    CASE VI_First_Fault_Source OF
        1: L_First_Fault_Source_Text := 'Heating';
        2: L_First_Fault_Source_Text := 'DHW';
        3: L_First_Fault_Source_Text := 'Ventilation';
        4: L_First_Fault_Source_Text := 'Lighting';
        5: L_First_Fault_Source_Text := 'Access';
        ELSE L_First_Fault_Source_Text := 'Unknown';
    END_CASE;

    L_Pending_Alarms[L_Pending_Count].Message := CONCAT('Diagnostics root cause: ', CONCAT(L_First_Fault_Source_Text, CONCAT(' / ', L_First_Fault_Type_Text)));
    L_Pending_Alarms[L_Pending_Count].Severity := E_ALERT_PRIORITY.ALERT_PRIORITY_HIGH;
    L_Pending_Alarms[L_Pending_Count].Is_Active := TRUE;
    L_Pending_Alarms[L_Pending_Count].Is_Acknowledged := FALSE;
END_IF;

FOR L_j := 1 TO GVL_CONSTANTS.C_MAX_BOILERS DO
    IF R_Trig_Boiler[L_j].Q AND L_Pending_Count < 10 THEN
        L_Pending_Count := L_Pending_Count + 1;
        L_Pending_Alarms[L_Pending_Count].Timestamp_MS := VI_System_Time_MS;
        L_Pending_Alarms[L_Pending_Count].Source := 'Boiler';
        L_Pending_Alarms[L_Pending_Count].Source_ID := TO_BYTE(L_j);
        L_Pending_Alarms[L_Pending_Count].Message := CONCAT('Авария котла №', INT_TO_STRING(L_j));
        L_Pending_Alarms[L_Pending_Count].Severity := E_ALERT_PRIORITY.ALERT_PRIORITY_HIGH;
        L_Pending_Alarms[L_Pending_Count].Is_Active := TRUE;
        L_Pending_Alarms[L_Pending_Count].Is_Acknowledged := FALSE;
    END_IF;
END_FOR;



// Обработка очереди новых тревог с учетом приоритетов
FOR L_i := 1 TO L_Pending_Count DO

    L_Target_Slot := 0;
    
    // 1. Ищем пустой слот
    FOR L_k := 1 TO GVL_CONSTANTS.C_MAX_ALARMS DO
        IF VO_Alarm_List[L_k].ID = 0 THEN
            L_Target_Slot := L_k;
            EXIT;
        END_IF;
    END_FOR;
    
    // 2. Ищем квитированную тревогу с наименьшим приоритетом
    IF L_Target_Slot = 0 THEN
        L_Min_Pri := 999;
        FOR L_k := 1 TO GVL_CONSTANTS.C_MAX_ALARMS DO
            IF VO_Alarm_List[L_k].Is_Acknowledged AND TO_INT(VO_Alarm_List[L_k].Severity) < L_Min_Pri THEN
                L_Min_Pri := TO_INT(VO_Alarm_List[L_k].Severity);
                L_Target_Slot := L_k;
            END_IF;
        END_FOR;
    END_IF;
    
    // 3. Ищем неквитированную тревогу с наименьшим приоритетом (если он ниже добавляемой)
    IF L_Target_Slot = 0 THEN
        L_Min_Pri := 999;
        FOR L_k := 1 TO GVL_CONSTANTS.C_MAX_ALARMS DO
            IF TO_INT(VO_Alarm_List[L_k].Severity) < L_Min_Pri AND TO_INT(VO_Alarm_List[L_k].Severity) < TO_INT(L_Pending_Alarms[L_i].Severity) THEN
                L_Min_Pri := TO_INT(VO_Alarm_List[L_k].Severity);
                L_Target_Slot := L_k;
            END_IF;
        END_FOR;
    END_IF;
    
    IF L_Target_Slot = 0 THEN 
        // Буфер полон критических неквитированных тревог. Не затираем!
        CONTINUE; 
    END_IF;
    
    VO_Alarm_List[L_Target_Slot] := L_Pending_Alarms[L_i];
    VO_Alarm_List[L_Target_Slot].ID := VIO_Next_Alarm_ID;
    VIO_Next_Alarm_ID := VIO_Next_Alarm_ID + 1;
    IF VIO_Next_Alarm_ID = 0 THEN VIO_Next_Alarm_ID := 1; END_IF;
    IF NOT L_Event_Pulse_Latched THEN
        VO_Event_Pulse := TRUE;
        VO_Event_Code := 1203;
        VO_Event_Value := TO_REAL(VO_Alarm_List[L_Target_Slot].Severity);
        L_Event_Pulse_Latched := TRUE;
    END_IF;
END_FOR;

// 3. Обновление статуса существующих тревог (ушли ли они?)
FOR L_i := 1 TO GVL_CONSTANTS.C_MAX_ALARMS DO
    IF VO_Alarm_List[L_i].ID <> 0 THEN
        IF VO_Alarm_List[L_i].Source = 'Gas' THEN VO_Alarm_List[L_i].Is_Active := VI_Gas_Alarm;
        ELSIF VO_Alarm_List[L_i].Source = 'Fire' THEN VO_Alarm_List[L_i].Is_Active := VI_Fire_Alarm;
        ELSIF VO_Alarm_List[L_i].Source = 'Flood' THEN VO_Alarm_List[L_i].Is_Active := VI_Flood_Alarm;
        ELSIF VO_Alarm_List[L_i].Source = 'Security' THEN VO_Alarm_List[L_i].Is_Active := VI_Security_Alarm;
        ELSIF VO_Alarm_List[L_i].Source = 'Diagnostics' THEN VO_Alarm_List[L_i].Is_Active := VI_First_Fault_Active;
        ELSIF VO_Alarm_List[L_i].Source = 'Boiler' THEN 
            IF TO_INT(VO_Alarm_List[L_i].Source_ID) >= 1 AND TO_INT(VO_Alarm_List[L_i].Source_ID) <= GVL_CONSTANTS.C_MAX_BOILERS THEN
                VO_Alarm_List[L_i].Is_Active := VI_Boiler_Errors[TO_INT(VO_Alarm_List[L_i].Source_ID)];
            END_IF;
        END_IF;
    END_IF;
END_FOR;

// 4. Квитирование тревог
IF VI_Acknowledge_All THEN
    FOR L_i := 1 TO GVL_CONSTANTS.C_MAX_ALARMS DO
        IF VO_Alarm_List[L_i].ID <> 0 THEN
            VO_Alarm_List[L_i].Is_Acknowledged := TRUE;
        END_IF;
    END_FOR;

    IF NOT L_Event_Pulse_Latched THEN
        VO_Event_Pulse := TRUE;
        VO_Event_Code := 1201;
        VO_Event_Value := TO_REAL(VO_Unacked_Count);
        L_Event_Pulse_Latched := TRUE;
    END_IF;
END_IF;

// 4.5 Автоквитирование некритичных тревог, если они больше не активны
FOR L_i := 1 TO GVL_CONSTANTS.C_MAX_ALARMS DO
    IF VO_Alarm_List[L_i].ID <> 0 AND NOT VO_Alarm_List[L_i].Is_Active AND NOT VO_Alarm_List[L_i].Is_Acknowledged THEN
        IF VO_Alarm_List[L_i].Severity <> E_ALERT_PRIORITY.ALERT_PRIORITY_CRITICAL THEN
            VO_Alarm_List[L_i].Is_Acknowledged := TRUE;
        END_IF;
    END_IF;
END_FOR;

// 5. Очистка списка (удаление неактивных И квитированных тревог)
// В кольцевом буфере мы просто помечаем слот как пустой (ID = 0), без сдвига массива
FOR L_i := 1 TO GVL_CONSTANTS.C_MAX_ALARMS DO
    IF VO_Alarm_List[L_i].ID <> 0 AND NOT VO_Alarm_List[L_i].Is_Active AND VO_Alarm_List[L_i].Is_Acknowledged THEN
        // Удаляем тревогу
        VO_Alarm_List[L_i].ID := 0;
        IF NOT L_Event_Pulse_Latched THEN
            VO_Event_Pulse := TRUE;
            VO_Event_Code := 1202;
            VO_Event_Value := 0.0;
            L_Event_Pulse_Latched := TRUE;
        END_IF;
    END_IF;
END_FOR;


// 6. Подсчет статистики и формирование глобальных флагов
VO_Global_Critical := FALSE;
VO_Global_Warning := FALSE;
VO_Siren_Active := FALSE;
VO_Active_Count := 0;
VO_Unacked_Count := 0;

FOR L_i := 1 TO GVL_CONSTANTS.C_MAX_ALARMS DO
    IF VO_Alarm_List[L_i].ID <> 0 THEN
        IF VO_Alarm_List[L_i].Is_Active THEN
            VO_Active_Count := VO_Active_Count + 1;
        END_IF;
        
        IF NOT VO_Alarm_List[L_i].Is_Acknowledged THEN
            VO_Unacked_Count := VO_Unacked_Count + 1;
            
            IF VO_Alarm_List[L_i].Severity = E_ALERT_PRIORITY.ALERT_PRIORITY_CRITICAL THEN
                VO_Global_Critical := TRUE;
                // Сирена работает только для неквитированных критических тревог, если не включен Mute
                IF NOT VI_Mute_Siren THEN
                    VO_Siren_Active := TRUE;
                END_IF;
            ELSIF VO_Alarm_List[L_i].Severity = E_ALERT_PRIORITY.ALERT_PRIORITY_HIGH THEN
                VO_Global_Warning := TRUE;
            END_IF;
        END_IF;
    END_IF;
END_FOR;
// >>> BULK_SYNC_ANCHOR: FB_Alarm_Manager <<<
          
END_FUNCTION_BLOCK

FUNCTION_BLOCK FB_Distributed_Recovery_Lock_Runtime
  VAR_INPUT
    VI_Enable : BOOL;
    VI_System_Time_MS : UDINT;
  END_VAR
  VAR
    L_Lock : ST_Distributed_Recovery_Lock;
    L_Finalized_Runtime_Continuity : BOOL;
  END_VAR

            IF NOT VI_Enable THEN
    GVL_Distributed_Recovery_Lock.G_Runtime_Valid := FALSE;
    RETURN;
END_IF;

L_Lock := GVL_Distributed_Recovery_Lock.G_Recovery_Lock;

L_Lock.Runtime_System_Time_MS := VI_System_Time_MS;
L_Lock.Lock_Valid := TRUE;

// Finalized runtime continuity proof chain.
L_Finalized_Runtime_Continuity :=
    GVL_SEMANTIC_PROGRESS.Semantic_Forward_Progress_Valid
    AND GVL_SEMANTIC_PROGRESS.Semantic_Execution_Continuity_OK
    AND NOT GVL_SEMANTIC_PROGRESS.Semantic_Progress_Lease_Expired
    AND NOT GVL_SEMANTIC_PROGRESS.Semantic_Progress_Quarantine_Active
    AND GVL_RUNTIME_SNAPSHOT.Snapshot_Frozen
    AND GVL_RUNTIME_SNAPSHOT.Snapshot_Publication_Allowed
    AND GVL_RUNTIME_SNAPSHOT.Snapshot_Copy_Valid
    AND GVL_RUNTIME_SNAPSHOT.Snapshot_Isolation_Valid
    AND NOT GVL_RUNTIME_SNAPSHOT.Snapshot_Mutation_Detected
    AND GVL_DISTRIBUTED_SNAPSHOT.Distributed_Publication_Reconciled
    AND GVL_DISTRIBUTED_SNAPSHOT.Distributed_Publication_Freeze_Valid
    AND GVL_DISTRIBUTED_SNAPSHOT.Distributed_Snapshot_Consistent
    AND GVL_DISTRIBUTED_COMMIT.Distributed_Commit_Valid
    AND GVL_DISTRIBUTED_COMMIT.Publication_Prepare_Valid
    AND GVL_DISTRIBUTED_COMMIT.Publication_Commit_Confirmed
    AND NOT GVL_DISTRIBUTED_COMMIT.Peer_Commit_Mismatch
    AND NOT GVL_DISTRIBUTED_COMMIT.Commit_Lease_Expired
    AND GVL_OUTPUT_EPOCH.Output_Publication_Valid
    AND GVL_OUTPUT_EPOCH.Output_Runtime_Epoch_Valid
    AND NOT GVL_OUTPUT_EPOCH.Output_Lease_Expired
    AND NOT GVL_OUTPUT_EPOCH.Output_Forced_Safe_Decay
    AND GVL_COMMAND_VERIFY.PreOutput_Barrier_OK
    AND NOT GVL_COMMAND_VERIFY.PreOutput_Block_IO;

// Cluster-exclusive recovery execution lock.
IF GVL_Distributed_Runtime.G_Split_Brain_Suspected
   OR GVL_Distributed_Projection_Ownership.G_Any_Ownership_Conflict
   OR GVL_Runtime_Sessions.G_Any_Stale_Session
   OR NOT L_Finalized_Runtime_Continuity THEN

    L_Lock.Lock_Conflict := TRUE;
    L_Lock.Distributed_Execution_Allowed := FALSE;

    GVL_Distributed_Recovery_Lock.G_Recovery_Execution_Blocked := TRUE;
    GVL_Distributed_Recovery_Lock.G_Rollback_Execution_Blocked := TRUE;
    GVL_Distributed_Recovery_Lock.G_Reopen_Execution_Blocked := TRUE;

    L_Lock.Status_Code := 3;
    L_Lock.Status_Text :=
        'Distributed recovery execution locked';

ELSE

    L_Lock.Recovery_Lock_Active := TRUE;
    L_Lock.Distributed_Execution_Allowed := TRUE;

    GVL_Distributed_Recovery_Lock.G_Recovery_Execution_Blocked := FALSE;
    GVL_Distributed_Recovery_Lock.G_Rollback_Execution_Blocked := FALSE;
    GVL_Distributed_Recovery_Lock.G_Reopen_Execution_Blocked := FALSE;

    L_Lock.Status_Code := 0;
    L_Lock.Status_Text :=
        'Distributed recovery lock healthy';

END_IF;

GVL_Distributed_Recovery_Lock.G_Recovery_Lock := L_Lock;

GVL_Distributed_Recovery_Lock.G_Runtime_Valid := TRUE;
GVL_Distributed_Recovery_Lock.G_Last_Update_MS :=
    VI_System_Time_MS;

GVL_Distributed_Recovery_Lock.G_Status_Code :=
    L_Lock.Status_Code;

GVL_Distributed_Recovery_Lock.G_Status_Text :=
    L_Lock.Status_Text;
          
END_FUNCTION_BLOCK

FUNCTION_BLOCK FB_Heating_Predictive_Controller
  VAR
    L_i : INT;
    L_Time_To_Heat : UDINT;
    L_Time_To_Comfort : UDINT;
    L_Now_TOD : UDINT;
  END_VAR

            // ==============================================================================
// Ownership note
// ------------------------------------------------------------------------------
// This block owns predictive preheat decision only.
// It does NOT modify thermal demand. Thermal demand is owned by
// FB_Heating_Thermal_Model and may be interpreted by downstream advisory layers.
// ==============================================================================

L_Now_TOD := GVL_TIME_SERVICE.G_Time_Of_Day_MS;

FOR L_i := 1 TO GVL_CONSTANTS.C_MAX_ZONES DO

    L_Time_To_Heat := GVL_HEATING_POLICY.G_Zone_Time_To_Heat_MS[L_i];
    L_Time_To_Comfort := GVL_HEATING_POLICY.G_Zone_Comfort_Time_MS[L_i];

    // Predictive preheat decision.
    IF GVL_HEATING_POLICY.G_Zone_Schedule_Enabled[L_i] THEN

        IF L_Time_To_Comfort > L_Now_TOD THEN
            IF (L_Time_To_Comfort - L_Now_TOD) <= L_Time_To_Heat THEN
                GVL_HEATING_POLICY.G_Zone_Preheat_Needed[L_i] := TRUE;
            ELSE
                GVL_HEATING_POLICY.G_Zone_Preheat_Needed[L_i] := FALSE;
            END_IF;
        END_IF;

    END_IF;

    // Confidence gating.
    IF GVL_HEATING_POLICY.G_Zone_Thermal_Model_Confidence[L_i] < 0.1 THEN
        GVL_HEATING_POLICY.G_Zone_Preheat_Needed[L_i] := FALSE;
    END_IF;

END_FOR;
          
END_FUNCTION_BLOCK

FUNCTION_BLOCK FB_System_Coordinator
  VAR_INPUT
    VI_Fire_Latched : BOOL;
    VI_Gas_Latched : BOOL;
    VI_Leak_Latched : BOOL;
    VI_IO_Degraded : BOOL;
    VI_Ownership_Violation : BOOL;
    VI_Behavior_Mode : E_Behavior_Mode;
  END_VAR
  VAR_OUTPUT
    VO_Block_Heating : BOOL;
    VO_Block_Ventilation : BOOL;
    VO_Block_Lighting : BOOL;
    VO_Block_Sockets : BOOL;
    VO_System_Degraded : BOOL;
    VO_Code : UDINT;
  END_VAR

            // reset
VO_Block_Heating := FALSE;
VO_Block_Ventilation := FALSE;
VO_Block_Lighting := FALSE;
VO_Block_Sockets := FALSE;
VO_System_Degraded := FALSE;
VO_Code := 0;

// FIRE has highest priority. Safety-stop ownership remains in PRG_Safety.
IF VI_Fire_Latched THEN
    VO_Block_Heating := TRUE;
    VO_Block_Ventilation := TRUE;
    VO_Block_Sockets := TRUE;
    VO_Code := 100;
    RETURN;
END_IF;

// GAS has higher priority than behavior mode.
IF VI_Gas_Latched THEN
    VO_Block_Heating := TRUE;
    VO_Block_Lighting := TRUE;
    VO_Block_Sockets := TRUE;
    VO_Code := 200;
    RETURN;
END_IF;

// LEAK blocks heating but does not suppress later degradation/mode overlays.
IF VI_Leak_Latched THEN
    VO_Block_Heating := TRUE;
    VO_Code := 300;
END_IF;

// IO degraded blocks heating and marks system degraded.
IF VI_IO_Degraded THEN
    VO_System_Degraded := TRUE;
    VO_Block_Heating := TRUE;
    IF VO_Code = 0 THEN
        VO_Code := 400;
    END_IF;
END_IF;

// Ownership violation marks system degraded. Test/result handler owns any safe-stop reaction.
IF VI_Ownership_Violation THEN
    VO_System_Degraded := TRUE;
    IF VO_Code = 0 THEN
        VO_Code := 500;
    END_IF;
END_IF;

// Behavior mode overlays. These are lower priority than safety/system faults.
CASE VI_Behavior_Mode OF
    BEHAVIOR_AWAY:
        VO_Block_Lighting := TRUE;
        VO_Block_Sockets := TRUE;
        IF VO_Code = 0 THEN
            VO_Code := 600;
        END_IF;

    BEHAVIOR_NIGHT:
        VO_Block_Lighting := TRUE;
        IF VO_Code = 0 THEN
            VO_Code := 700;
        END_IF;

    BEHAVIOR_MAINTENANCE:
        VO_Block_Heating := TRUE;
        VO_Block_Ventilation := TRUE;
        IF VO_Code = 0 THEN
            VO_Code := 800;
        END_IF;
ELSE
        // No fallback required
END_CASE;
          
END_FUNCTION_BLOCK

FUNCTION_BLOCK FB_Water_Isolation_Path_Resolver
  VAR_INPUT
    VI_Enable : BOOL;
    VI_System_Time_MS : UDINT;
  END_VAR
  VAR
    L_i : INT;
    L_Edge : ST_Water_Hydraulic_Topology_Edge;
    L_Path : ST_Water_Isolation_Path_Runtime_State;
    L_Validation : ST_Water_Topology_Validation_State;
    L_Any_Shared_Trunk : BOOL;
    L_Any_Conflict : BOOL;
    L_Any_Fallback : BOOL;
  END_VAR

            IF NOT VI_Enable THEN
    GVL_Water_Hydraulic_Graph.G_Runtime_Valid := FALSE;
    RETURN;
END_IF;

FOR L_i := 1 TO GVL_CONSTANTS.C_MAX_FLOOD_SENSORS DO

    L_Validation :=
        GVL_Water_Topology_Validation.G_Validation_State[L_i];

    // Graph edge publication.
    L_Edge := (Runtime_Valid := TRUE);

    L_Edge.Edge_Id := TO_UINT(L_i);

    L_Edge.Upstream_Segment_Id :=
        GVL_Water_Hydraulic_Topology.G_Topology_Node[L_i].Hydraulic_Segment_Id;

    L_Edge.Downstream_Segment_Id :=
        GVL_Water_Hydraulic_Topology.G_Topology_Node[L_i].Hydraulic_Zone_Id;

    L_Edge.Isolation_Group_Id :=
        GVL_Water_Hydraulic_Topology.G_Topology_Node[L_i].Isolation_Group_Id;

    L_Edge.Valve_Group_Id :=
        GVL_Water_Hydraulic_Topology.G_Topology_Node[L_i].Valve_Group_Id;

    // Shared trunk semantics.
    IF L_Edge.Valve_Group_Id = 3 THEN
        L_Edge.Shared_Trunk := TRUE;
        L_Edge.Cross_Zone_Dependency := TRUE;
    END_IF;

    L_Edge.Dependency_Valid :=
        L_Validation.Topology_Valid;

    L_Edge.Dependency_Ambiguous :=
        L_Validation.Topology_Ambiguous;

    L_Edge.Selective_Isolation_Allowed :=
        L_Validation.Selective_Isolation_Allowed;

    L_Edge.Global_Fallback_Required :=
        L_Validation.Global_Fallback_Required;

    // Isolation path runtime.
    L_Path := (Runtime_Valid := TRUE);

    L_Path.Runtime_System_Time_MS :=
        VI_System_Time_MS;

    L_Path.Sensor_Id := TO_UINT(L_i);

    L_Path.Isolation_Path_Valid :=
        L_Edge.Dependency_Valid;

    L_Path.Isolation_Path_Ambiguous :=
        L_Edge.Dependency_Ambiguous;

    L_Path.Active_Isolation_Group_Id :=
        L_Edge.Isolation_Group_Id;

    L_Path.Active_Valve_Group_Id :=
        L_Edge.Valve_Group_Id;

    L_Path.Shared_Trunk_Impact :=
        L_Edge.Shared_Trunk;

    L_Path.Cross_Zone_Impact :=
        L_Edge.Cross_Zone_Dependency;

    L_Path.Selective_Isolation_Allowed :=
        L_Edge.Selective_Isolation_Allowed;

    L_Path.Global_Fallback_Required :=
        L_Edge.Global_Fallback_Required;

    // Multi-valve/shared-trunk path.
    IF L_Path.Shared_Trunk_Impact THEN
        L_Path.Multi_Valve_Path := TRUE;
    END_IF;

    // Conflict detection.
    IF L_Path.Isolation_Path_Ambiguous THEN
        L_Path.Conflict_Detected := TRUE;
    END_IF;

    // Conservative escalation.
    IF L_Path.Conflict_Detected THEN
        L_Path.Global_Fallback_Required := TRUE;
        L_Path.Selective_Isolation_Allowed := FALSE;

        L_Path.Status_Code := 2;
        L_Path.Status_Text :=
            'Isolation path conflict detected';

    ELSIF L_Path.Shared_Trunk_Impact THEN
        L_Path.Status_Code := 1;
        L_Path.Status_Text :=
            'Shared trunk isolation path active';

    ELSE
        L_Path.Status_Code := 0;
        L_Path.Status_Text :=
            'Isolation path resolved';
    END_IF;

    GVL_Water_Hydraulic_Graph.G_Topology_Edge[L_i] :=
        L_Edge;

    GVL_Water_Hydraulic_Graph.G_Isolation_Path[L_i] :=
        L_Path;

    L_Any_Shared_Trunk :=
        L_Any_Shared_Trunk
        OR L_Path.Shared_Trunk_Impact;

    L_Any_Conflict :=
        L_Any_Conflict
        OR L_Path.Conflict_Detected;

    L_Any_Fallback :=
        L_Any_Fallback
        OR L_Path.Global_Fallback_Required;

END_FOR;

GVL_Water_Hydraulic_Graph.G_Any_Shared_Trunk :=
    L_Any_Shared_Trunk;

GVL_Water_Hydraulic_Graph.G_Any_Conflict :=
    L_Any_Conflict;

GVL_Water_Hydraulic_Graph.G_Any_Global_Fallback_Required :=
    L_Any_Fallback;

GVL_Water_Hydraulic_Graph.G_Runtime_Valid := TRUE;
GVL_Water_Hydraulic_Graph.G_Last_Update_MS := VI_System_Time_MS;

IF L_Any_Conflict THEN
    GVL_Water_Hydraulic_Graph.G_Status_Code := 2;
    GVL_Water_Hydraulic_Graph.G_Status_Text :=
        'Hydraulic graph conflicts detected';
ELSIF L_Any_Shared_Trunk THEN
    GVL_Water_Hydraulic_Graph.G_Status_Code := 1;
    GVL_Water_Hydraulic_Graph.G_Status_Text :=
        'Shared trunk governance active';
ELSE
    GVL_Water_Hydraulic_Graph.G_Status_Code := 0;
    GVL_Water_Hydraulic_Graph.G_Status_Text :=
        'Hydraulic graph runtime healthy';
END_IF;
          
END_FUNCTION_BLOCK

FUNCTION_BLOCK FB_Ownership_Watchdog
  VAR_INPUT
    VI_Gas_Level : REAL;
    VI_Gas_Alarm : BOOL;
    VI_Leak_Alarm : BOOL;
    VI_Smoke_Alarm : BOOL;
  END_VAR
  VAR_OUTPUT
    VO_Ownership_Violation : BOOL;
  END_VAR
  VAR
    L_Last_Gas_Alarm : BOOL;
    L_Last_Leak_Alarm : BOOL;
    L_Last_Smoke_Alarm : BOOL;
  END_VAR

            VO_Ownership_Violation := FALSE;

// Gas: signal present, alarm disappeared
IF (VI_Gas_Level > 20.0) AND L_Last_Gas_Alarm AND (NOT VI_Gas_Alarm) THEN
    VO_Ownership_Violation := TRUE;
END_IF;

// Leak: once latched should not drop instantly
IF L_Last_Leak_Alarm AND (NOT VI_Leak_Alarm) THEN
    VO_Ownership_Violation := TRUE;
END_IF;

// Smoke: same rule
IF L_Last_Smoke_Alarm AND (NOT VI_Smoke_Alarm) THEN
    VO_Ownership_Violation := TRUE;
END_IF;

L_Last_Gas_Alarm := VI_Gas_Alarm;
L_Last_Leak_Alarm := VI_Leak_Alarm;
L_Last_Smoke_Alarm := VI_Smoke_Alarm;
          
END_FUNCTION_BLOCK

FUNCTION_BLOCK FB_Valve_Test_Manager
  VAR_INPUT
    VI_System_Time_MS : UDINT;
    VI_IsActivePLC : BOOL;
  END_VAR
  VAR_OUTPUT
    VO_Test_Active : BOOL;
    VO_Current_Valve : INT;
    VO_Valve_Cmd : ARRAY[1..GVL_CONSTANTS.C_MAX_MANIFOLDS] OF BOOL;
    VO_Test_Results : ARRAY[1..GVL_CONSTANTS.C_MAX_MANIFOLDS] OF BOOL;
    VO_Status_Msg : STRING(200);
  END_VAR
  VAR_IN_OUT
    VI_Valve_Currents : ARRAY[1..GVL_CONSTANTS.C_MAX_MANIFOLDS] OF REAL;
    VI_Valve_End_Switches : ARRAY[1..GVL_CONSTANTS.C_MAX_MANIFOLDS] OF BOOL;
    VI_Config : ARRAY[1..GVL_CONSTANTS.C_MAX_MANIFOLDS] OF ST_Valve_Test_Config;
  END_VAR
  VAR
    L_State : INT;
    L_Current_Valve : INT := 1;
    L_Test_Start_Time : UDINT;
    L_Last_Test_Time : ARRAY[1..GVL_CONSTANTS.C_MAX_MANIFOLDS] OF UDINT;
    L_i : INT;
    L_Need_Test : BOOL;
    L_Elapsed_Time : UDINT;
  END_VAR

            IF NOT VI_IsActivePLC THEN RETURN; END_IF;

CASE L_State OF
    0: // Ожидание
        VO_Test_Active := FALSE;
        L_Need_Test := FALSE;
        
        // Поиск клапана, которому нужен тест (раз в неделю)
        FOR L_i := 1 TO GVL_CONSTANTS.C_MAX_MANIFOLDS DO
            IF VI_Config[L_i].enabled AND ((VI_System_Time_MS - L_Last_Test_Time[L_i]) > (VI_Config[L_i].test_interval_days * 86400000)) THEN
                L_Current_Valve := L_i;
                L_Need_Test := TRUE;
                EXIT;
            END_IF;
        END_FOR;
        
        IF L_Need_Test THEN
            L_State := 1;
            L_Test_Start_Time := VI_System_Time_MS;
            VO_Test_Active := TRUE;
            VO_Current_Valve := L_Current_Valve;
            VO_Valve_Cmd[L_Current_Valve] := TRUE; // Открываем
            VO_Status_Msg := CONCAT('ТЕСТ КЛАПАНА ', INT_TO_STRING(L_Current_Valve));
            VO_Test_Results[L_Current_Valve] := TRUE; // Сброс результата
        END_IF;
        
    1: // Тестирование (ожидание открытия)
        L_Elapsed_Time := (VI_System_Time_MS - L_Test_Start_Time);
        
        IF VI_Valve_End_Switches[L_Current_Valve] THEN
            // Концевик сработал до истечения таймаута
            // Проверка тока
            IF ABS(VI_Valve_Currents[L_Current_Valve] - VI_Config[L_Current_Valve].Nominal_Current) > (VI_Config[L_Current_Valve].Nominal_Current * 0.2) THEN
                VO_Test_Results[L_Current_Valve] := FALSE; // Ошибка по току
            END_IF;
            
            GVL_Retain.G_Valve_Test_Results[L_Current_Valve] := VO_Test_Results[L_Current_Valve];
            
            VO_Valve_Cmd[L_Current_Valve] := FALSE; // Закрываем
            L_Test_Start_Time := VI_System_Time_MS; // Перезапускаем таймер для проверки закрытия
            L_State := 2;
        ELSIF L_Elapsed_Time > TO_UDINT(VI_Config[L_Current_Valve].nominal_close_time_sec * 1000.0) THEN
            // Таймаут открытия (заклинивание)
            VO_Test_Results[L_Current_Valve] := FALSE; 
            GVL_Retain.G_Valve_Test_Results[L_Current_Valve] := FALSE;
            VO_Status_Msg := CONCAT('ОШИБКА: ЗАКЛИНИВАНИЕ КЛАПАНА ', INT_TO_STRING(L_Current_Valve));
            
            VO_Valve_Cmd[L_Current_Valve] := FALSE; // Закрываем
            L_Test_Start_Time := VI_System_Time_MS; // Перезапускаем таймер
            L_State := 2;
        END_IF;
        
    2: // Ожидание закрытия
        L_Elapsed_Time := (VI_System_Time_MS - L_Test_Start_Time);
        
        IF NOT VI_Valve_End_Switches[L_Current_Valve] THEN
            // Концевик разомкнулся (клапан закрыт)
            L_Last_Test_Time[L_Current_Valve] := VI_System_Time_MS;
            L_State := 0;
            IF VO_Test_Results[L_Current_Valve] THEN
                VO_Status_Msg := 'ТЕСТ ЗАВЕРШЕН УСПЕШНО';
            END_IF;
        ELSIF L_Elapsed_Time > TO_UDINT(VI_Config[L_Current_Valve].nominal_close_time_sec * 1000.0) THEN
            // Таймаут закрытия (заклинивание)
            VO_Test_Results[L_Current_Valve] := FALSE; 
            GVL_Retain.G_Valve_Test_Results[L_Current_Valve] := FALSE;
            VO_Status_Msg := CONCAT('ОШИБКА: НЕ ЗАКРЫЛСЯ КЛАПАН ', INT_TO_STRING(L_Current_Valve));
            
            L_Last_Test_Time[L_Current_Valve] := VI_System_Time_MS;
            L_State := 0;
        END_IF;
ELSE
        // No fallback required
END_CASE;
          
END_FUNCTION_BLOCK

FUNCTION_BLOCK FB_PID_Controller
  VAR_INPUT
    VI_SetPoint : REAL;
    VI_ProcessValue : REAL;
    VI_Kp : REAL;
    VI_Tn : REAL;
    VI_Tv : REAL;
    VI_Y_Min : REAL := REAL#0.0;
    VI_Y_Max : REAL := REAL#100.0;
    VI_Manual_Mode : BOOL;
    VI_Manual_Value : REAL;
    VI_Deadband : REAL := REAL#0.1;
    VI_Cycle_Time_S : REAL := REAL#0.01;
    VI_Reset : BOOL;
  END_VAR
  VAR_OUTPUT
    VO_Output : REAL;
    VO_Error : REAL;
    VO_Limiting : BOOL;
  END_VAR
  VAR
    L_Integral_Sum : REAL;
    L_Prev_Error : REAL;
    L_Derivative : REAL;
    L_P_Term : REAL;
    L_I_Candidate : REAL;
    L_D_Term : REAL;
    L_Output_Predicted : REAL;
    L_Output_Raw : REAL;
    L_Cycle_Time_Safe : REAL;
  END_VAR

            L_Cycle_Time_Safe := VI_Cycle_Time_S;
IF L_Cycle_Time_Safe <= REAL#0.0 THEN
    L_Cycle_Time_Safe := REAL#0.01;
END_IF;

VO_Error := VI_SetPoint - VI_ProcessValue;
IF ABS(VO_Error) < VI_Deadband THEN
    VO_Error := REAL#0.0;
END_IF;

IF VI_Reset THEN
    L_Integral_Sum := REAL#0.0;
    L_Prev_Error := REAL#0.0;
    VO_Output := LIMIT(VI_Y_Min, REAL#0.0, VI_Y_Max);
    VO_Limiting := FALSE;
    RETURN;
END_IF;

L_P_Term := VI_Kp * VO_Error;

IF VI_Tv > REAL#0.0 THEN
    L_Derivative := (VO_Error - L_Prev_Error) / L_Cycle_Time_Safe;
    L_D_Term := VI_Kp * VI_Tv * L_Derivative;
ELSE
    L_Derivative := REAL#0.0;
    L_D_Term := REAL#0.0;
END_IF;

IF VI_Manual_Mode THEN
    VO_Output := LIMIT(VI_Y_Min, VI_Manual_Value, VI_Y_Max);
    L_Integral_Sum := VO_Output - L_P_Term - L_D_Term;
    L_Prev_Error := VO_Error;
    VO_Limiting := (VO_Output <= VI_Y_Min) OR (VO_Output >= VI_Y_Max);
    RETURN;
END_IF;

IF VI_Tn > REAL#0.0 THEN
    L_I_Candidate := L_Integral_Sum + ((VI_Kp / VI_Tn) * VO_Error * L_Cycle_Time_Safe);
ELSE
    L_I_Candidate := L_Integral_Sum;
END_IF;

L_Output_Predicted := L_P_Term + L_I_Candidate + L_D_Term;

// Anti-windup: accept the new integral only if it does not push the output farther into saturation.
IF VI_Tn > REAL#0.0 THEN
    IF (L_Output_Predicted > VI_Y_Max) AND (VO_Error > REAL#0.0) THEN
        // hold integral
    ELSIF (L_Output_Predicted < VI_Y_Min) AND (VO_Error < REAL#0.0) THEN
        // hold integral
    ELSE
        L_Integral_Sum := L_I_Candidate;
    END_IF;
END_IF;

L_Output_Raw := L_P_Term + L_Integral_Sum + L_D_Term;
VO_Output := LIMIT(VI_Y_Min, L_Output_Raw, VI_Y_Max);
VO_Limiting := (L_Output_Raw > VI_Y_Max) OR (L_Output_Raw < VI_Y_Min);
L_Prev_Error := VO_Error;

// >>> BULK_SYNC_ANCHOR: FB_PID_Controller <<<
          
END_FUNCTION_BLOCK

FUNCTION_BLOCK FB_ADS_Runtime_Adapter
  VAR_INPUT
    VI_Enable : BOOL;
    VI_System_Time_MS : UDINT;
  END_VAR
  VAR
    L_Frame : ST_Runtime_Bus_Frame;
    L_TX_Index : UINT;
  END_VAR

            IF NOT VI_Enable THEN
    RETURN;
END_IF;

L_TX_Index := UDINT_TO_UINT(GVL_Runtime_Bus.G_Last_Sequence_Id);

IF (L_TX_Index >= 1)
   AND (L_TX_Index <= 128) THEN

    L_Frame := GVL_Runtime_Bus.G_TX_Frames[L_TX_Index];

    IF L_Frame.Frame_Valid THEN

        IF GVL_Distributed_Authority.G_Distributed_Safety_Barrier_OK
           AND GVL_Runtime_Sessions.G_Runtime_Valid
           AND NOT GVL_Runtime_Sessions.G_Any_Stale_Session
           AND NOT GVL_Runtime_Sessions.G_Any_Quarantined_Session THEN

            L_Frame.Frame_Ack_Received := TRUE;
            L_Frame.Replication_Consistent := TRUE;
            L_Frame.Replication_Rejected := FALSE;
            L_Frame.Status_Code := 0;

        ELSE

            L_Frame.Frame_Ack_Received := FALSE;
            L_Frame.Replication_Consistent := FALSE;
            L_Frame.Replication_Rejected := TRUE;
            L_Frame.Status_Code := 2;

        END_IF;

        GVL_Runtime_Bus.G_TX_Frames[L_TX_Index] := L_Frame;
        GVL_Runtime_Bus.G_TX_Healthy := L_Frame.Replication_Consistent;
        GVL_Runtime_Bus.G_Any_Replication_Rejected := L_Frame.Replication_Rejected;

    END_IF;

END_IF;
          
END_FUNCTION_BLOCK

FUNCTION_BLOCK FB_Diagnostics_Event_Manager
  VAR_INPUT
    VI_Code : UDINT;
    VI_Severity : INT;
    VI_Active : BOOL;
    VI_Timestamp : UDINT;
    VI_Source : INT;
  END_VAR
  VAR_IN_OUT
    VIO_Events : ARRAY[1..50] OF ST_Diagnostic_Event;
    VIO_Count : INT;
  END_VAR
  VAR
    L_Index : INT;
    L_i : INT;
    L_Found_Index : INT;
    L_Was_Active : BOOL;
    L_Debounce_Index : INT;
    L_Oldest_Index : INT;
    L_Oldest_Time : UDINT;
    L_Stable_State : BOOL;
    L_Debounce_Used : ARRAY[1..50] OF BOOL;
    L_Debounce_Code : ARRAY[1..50] OF UDINT;
    L_Debounce_Source : ARRAY[1..50] OF INT;
    L_Debounce_Last_Input_State : ARRAY[1..50] OF BOOL;
    L_Debounce_Stable_State : ARRAY[1..50] OF BOOL;
    L_Debounce_Last_Change_Time : ARRAY[1..50] OF UDINT;
  END_VAR

            L_Found_Index := 0;
L_Was_Active := FALSE;
FOR L_i := 1 TO 50 DO
    IF (VIO_Events[L_i].Code = VI_Code) AND (VIO_Events[L_i].Source = VI_Source) THEN
        L_Found_Index := L_i;
        L_Was_Active := VIO_Events[L_i].Active;
        EXIT;
    END_IF;
END_FOR;

L_Debounce_Index := 0;
L_Oldest_Time := 16#FFFFFFFF;
L_Oldest_Index := 1;

FOR L_i := 1 TO 50 DO
    IF L_Debounce_Used[L_i] THEN
        IF (L_Debounce_Code[L_i] = VI_Code) AND (L_Debounce_Source[L_i] = VI_Source) THEN
            L_Debounce_Index := L_i;
            EXIT;
        END_IF;
        IF L_Debounce_Last_Change_Time[L_i] < L_Oldest_Time THEN
            L_Oldest_Time := L_Debounce_Last_Change_Time[L_i];
            L_Oldest_Index := L_i;
        END_IF;
    ELSE
        L_Debounce_Index := L_i;
        EXIT;
    END_IF;
END_FOR;

IF L_Debounce_Index = 0 THEN
    L_Debounce_Index := L_Oldest_Index;
END_IF;

IF NOT L_Debounce_Used[L_Debounce_Index] OR
   (L_Debounce_Code[L_Debounce_Index] <> VI_Code) OR
   (L_Debounce_Source[L_Debounce_Index] <> VI_Source) THEN
    L_Debounce_Used[L_Debounce_Index] := TRUE;
    L_Debounce_Code[L_Debounce_Index] := VI_Code;
    L_Debounce_Source[L_Debounce_Index] := VI_Source;
    L_Debounce_Last_Input_State[L_Debounce_Index] := VI_Active;
    L_Debounce_Stable_State[L_Debounce_Index] := FALSE;
    L_Debounce_Last_Change_Time[L_Debounce_Index] := VI_Timestamp;
END_IF;

IF VI_Active <> L_Debounce_Last_Input_State[L_Debounce_Index] THEN
    L_Debounce_Last_Input_State[L_Debounce_Index] := VI_Active;
    L_Debounce_Last_Change_Time[L_Debounce_Index] := VI_Timestamp;
END_IF;

IF (VI_Timestamp - L_Debounce_Last_Change_Time[L_Debounce_Index]) > 2000 THEN
    L_Debounce_Stable_State[L_Debounce_Index] := L_Debounce_Last_Input_State[L_Debounce_Index];
END_IF;

L_Stable_State := L_Debounce_Stable_State[L_Debounce_Index];

IF L_Stable_State THEN
    IF NOT L_Was_Active THEN
        L_Index := (VIO_Count MOD 50) + 1;
        VIO_Events[L_Index].Code := VI_Code;
        VIO_Events[L_Index].Severity := VI_Severity;
        VIO_Events[L_Index].Active := TRUE;
        VIO_Events[L_Index].Timestamp := VI_Timestamp;
        VIO_Events[L_Index].Source := VI_Source;
        VIO_Count := VIO_Count + 1;
    ELSIF L_Found_Index > 0 THEN
        VIO_Events[L_Found_Index].Severity := VI_Severity;
    END_IF;
ELSE
    IF L_Found_Index > 0 THEN
        VIO_Events[L_Found_Index].Active := FALSE;
    END_IF;
END_IF;

// >>> BULK_SYNC_ANCHOR: FB_Diagnostics_Event_Manager <<<
          
END_FUNCTION_BLOCK

FUNCTION_BLOCK FB_Water_Valve_Runtime_Governance
  VAR_INPUT
    VI_Enable : BOOL;
    VI_System_Time_MS : UDINT;
  END_VAR
  VAR
    L_i : INT;
    L_Authority : ST_Water_Isolation_Authority_State;
    L_Valve : ST_Water_Valve_Runtime_State;
    L_Any_Degraded : BOOL;
    L_Any_Confirmation_Unknown : BOOL;
    L_Any_Unsafe_Reopen : BOOL;
  END_VAR

            IF NOT VI_Enable THEN
    GVL_Water_Valve_Runtime.G_Runtime_Valid := FALSE;
    RETURN;
END_IF;

FOR L_i := 1 TO GVL_CONSTANTS.C_MAX_FLOOD_SENSORS DO

    L_Authority :=
        GVL_Water_Isolation_Authority.G_Authority_State[L_i];

    L_Valve := (Runtime_Valid := TRUE);

    L_Valve.Runtime_System_Time_MS := VI_System_Time_MS;

    L_Valve.Valve_Id := L_Authority.Valve_Group_Id;
    L_Valve.Valve_Group_Id := L_Authority.Valve_Group_Id;

    L_Valve.Close_Requested :=
        L_Authority.Selective_Authority_Allowed
        OR L_Authority.Global_Fallback_Required;

    L_Valve.Global_Fallback_Request :=
        L_Authority.Global_Fallback_Required;

    L_Valve.Selective_Authority_Allowed :=
        L_Authority.Selective_Authority_Allowed;

    // Observe-only compatibility visibility.
    L_Valve.Physical_Output_Active :=
        GVL_COMMAND_SHADOW.G_Close_Valve_35
        OR GVL_COMMAND_SHADOW.G_Close_Valve_36;

    L_Valve.Output_Command_Projected :=
        L_Valve.Close_Requested;

    // Feedback/runtime hooks.
    L_Valve.Confirmation_Available :=
        GVL_Water_Valve_Feedback.G_Valve_Feedback_State[L_i].Feedback_Available;

    IF L_Valve.Confirmation_Available THEN

        L_Valve.Confirmed_Closed :=
            GVL_Water_Valve_Feedback.G_Valve_Feedback_State[L_i].Confirmed_Closed;

    ELSE

        L_Valve.Confirmation_Unknown := TRUE;

    END_IF;

    // Observe-only semantics must not force degraded state.
    L_Valve.Diagnostics_Available := FALSE;
    L_Valve.Valve_Healthy := TRUE;

    IF L_Valve.Confirmation_Available
       AND NOT L_Valve.Confirmed_Closed
       AND L_Valve.Close_Requested THEN

        L_Valve.Valve_Degraded := TRUE;

    END_IF;

    IF L_Valve.Valve_Degraded THEN

        L_Valve.Unsafe_Reopen_Denied := TRUE;
        L_Valve.Recovery_Allowed := FALSE;

        L_Valve.Status_Code := 2;
        L_Valve.Status_Text :=
            'Recovery denied: valve degraded';

    ELSIF L_Valve.Confirmation_Unknown THEN

        L_Valve.Status_Code := 1;
        L_Valve.Status_Text :=
            'Valve confirmation unavailable';

    ELSE

        L_Valve.Status_Code := 0;
        L_Valve.Status_Text :=
            'Valve governance runtime healthy';

    END_IF;

    GVL_Water_Valve_Runtime.G_Valve_Runtime_State[L_i] :=
        L_Valve;

    L_Any_Degraded :=
        L_Any_Degraded
        OR L_Valve.Valve_Degraded;

    L_Any_Confirmation_Unknown :=
        L_Any_Confirmation_Unknown
        OR L_Valve.Confirmation_Unknown;

    L_Any_Unsafe_Reopen :=
        L_Any_Unsafe_Reopen
        OR L_Valve.Unsafe_Reopen_Denied;

END_FOR;

GVL_Water_Valve_Runtime.G_Any_Valve_Degraded :=
    L_Any_Degraded;

GVL_Water_Valve_Runtime.G_Any_Confirmation_Unknown :=
    L_Any_Confirmation_Unknown;

GVL_Water_Valve_Runtime.G_Any_Unsafe_Reopen_Denied :=
    L_Any_Unsafe_Reopen;

GVL_Water_Valve_Runtime.G_Runtime_Valid := TRUE;
GVL_Water_Valve_Runtime.G_Last_Update_MS := VI_System_Time_MS;

IF L_Any_Degraded THEN
    GVL_Water_Valve_Runtime.G_Status_Code := 2;
    GVL_Water_Valve_Runtime.G_Status_Text :=
        'Valve governance degraded';
ELSIF L_Any_Confirmation_Unknown THEN
    GVL_Water_Valve_Runtime.G_Status_Code := 1;
    GVL_Water_Valve_Runtime.G_Status_Text :=
        'Valve confirmation unknown';
ELSE
    GVL_Water_Valve_Runtime.G_Status_Code := 0;
    GVL_Water_Valve_Runtime.G_Status_Text :=
        'Valve governance runtime active';
END_IF;
          
END_FUNCTION_BLOCK

FUNCTION_BLOCK FB_Water_Output_Reconciliation
  VAR_INPUT
    VI_Enable : BOOL;
    VI_System_Time_MS : UDINT;
  END_VAR
  VAR
    L_i : INT;
    L_Output : ST_Water_Output_Projection_State;
    L_Valve : ST_Water_Valve_Runtime_State;
    L_State : ST_Water_Output_Reconciliation_State;
    L_Any_Runtime_Mismatch : BOOL;
    L_Any_Confirmation_Mismatch : BOOL;
    L_Any_Conflict : BOOL;
  END_VAR

            IF NOT VI_Enable THEN
    GVL_Water_Output_Reconciliation.G_Runtime_Valid := FALSE;
    RETURN;
END_IF;

FOR L_i := 1 TO GVL_CONSTANTS.C_MAX_FLOOD_SENSORS DO

    L_Output := GVL_Water_Output_Projection.G_Output_Projection_State[L_i];
    L_Valve := GVL_Water_Valve_Runtime.G_Valve_Runtime_State[L_i];

    L_State.Runtime_Valid := TRUE;
    L_State.Runtime_System_Time_MS := VI_System_Time_MS;

    L_State.Valve_Group_Id := L_Output.Valve_Group_Id;
    L_State.Projection_Active := L_Output.Physical_Close_Project;
    L_State.Runtime_Output_Active := L_Valve.Physical_Output_Active;
    L_State.Expected_Closed := L_Output.Expected_Closed;
    L_State.Confirmed_Closed := L_Valve.Confirmed_Closed;
    L_State.Confirmation_Unknown := L_Valve.Confirmation_Unknown;

    IF L_Valve.Confirmation_Available THEN

        IF L_State.Projection_Active <> L_State.Runtime_Output_Active THEN
            L_State.Projection_Runtime_Mismatch := TRUE;
        END_IF;

        IF L_State.Expected_Closed
           AND NOT L_State.Confirmed_Closed THEN
            L_State.Projection_Confirmation_Mismatch := TRUE;
        END_IF;

    END_IF;

    IF L_Output.Projection_Allowed
       AND L_Output.Projection_Denied THEN
        L_State.Conflict_Detected := TRUE;
    END_IF;

    IF L_Output.Valve_Group_Id = 0 THEN
        L_State.Topology_Invalid := TRUE;
    END_IF;

    L_State.Reconciliation_Healthy :=
        NOT L_State.Projection_Runtime_Mismatch
        AND NOT L_State.Projection_Confirmation_Mismatch
        AND NOT L_State.Conflict_Detected
        AND NOT L_State.Topology_Invalid;

    IF L_State.Conflict_Detected THEN
        L_State.Status_Code := 3;
        L_State.Status_Text := 'Projection conflict detected';
    ELSIF L_State.Projection_Runtime_Mismatch THEN
        L_State.Status_Code := 2;
        L_State.Status_Text := 'Projection runtime mismatch';
    ELSIF L_State.Projection_Confirmation_Mismatch THEN
        L_State.Status_Code := 1;
        L_State.Status_Text := 'Projection confirmation mismatch';
    ELSE
        L_State.Status_Code := 0;
        L_State.Status_Text := 'Reconciliation healthy';
    END_IF;

    GVL_Water_Output_Reconciliation.G_Reconciliation_State[L_i] := L_State;
END_FOR;
          
END_FUNCTION_BLOCK

FUNCTION_BLOCK FB_Sensor_Analog_Processing
  VAR_INPUT
    VI_Raw_Value : WORD;
    VI_Sensor_Type : INT := 0;
    VI_Min_Scale : REAL;
    VI_Max_Scale : REAL;
    VI_Offset : REAL;
    VI_Multiplier : REAL := 1.0;
    VI_Filter_Time_MS : UDINT := GVL_CONSTANTS.C_MS_IN_SECOND;
    VI_System_Time_MS : UDINT;
    VI_Fallback_Mode : INT := 0;
    VI_Default_Value : REAL := 0.0;
  END_VAR
  VAR_OUTPUT
    VO_Value : REAL;
    VO_Error : BOOL;
    VO_Diag_Code : WORD;
  END_VAR
  VAR
    L_Scaled : REAL;
    L_Filtered : REAL;
    L_History : ARRAY[0..9] OF REAL;
    L_History_Idx : INT := 0;
    L_History_Sum : REAL := 0.0;
    L_History_Count : INT := 0;
    L_Last_Time : UDINT;
    L_DT : UDINT;
    L_First_Scan : BOOL := TRUE;
    L_i : INT;
  END_VAR

            // 1. Error checking and scaling based on sensor type
VO_Error := FALSE;
VO_Diag_Code := 0;

CASE VI_Sensor_Type OF
    0: // 4-20mA (NAMUR NE43: < 3.6mA or > 21mA)
        IF VI_Raw_Value < GVL_CONSTANTS.C_ANALOG_3_6MA_RAW THEN // < 3.6mA (Open circuit)
            VO_Error := TRUE;
            VO_Diag_Code := 1;
        ELSIF VI_Raw_Value > GVL_CONSTANTS.C_ANALOG_21MA_RAW THEN // > 21mA (Short circuit)
            VO_Error := TRUE;
            VO_Diag_Code := 2;
        ELSE
            // 4mA = 5529, 20mA = 27648
            L_Scaled := VI_Min_Scale + (TO_REAL(VI_Raw_Value - GVL_CONSTANTS.C_ANALOG_4MA_RAW) / TO_REAL(GVL_CONSTANTS.C_ANALOG_RAW_MAX - GVL_CONSTANTS.C_ANALOG_4MA_RAW)) * (VI_Max_Scale - VI_Min_Scale);
        END_IF;
        
    1: // 0-10V (0-27648)
        IF VI_Raw_Value > GVL_CONSTANTS.C_ANALOG_10V_MAX_RAW THEN // Out of range
            VO_Error := TRUE;
            VO_Diag_Code := 3;
        ELSE
            L_Scaled := VI_Min_Scale + (TO_REAL(VI_Raw_Value) / TO_REAL(GVL_CONSTANTS.C_ANALOG_RAW_MAX)) * (VI_Max_Scale - VI_Min_Scale);
        END_IF;
        
    2: // PT100/1000 (Direct temperature * 10, e.g., 255 = 25.5C)
        // Typically, 16-bit signed integer for temperature
        IF VI_Raw_Value = 16#7FFF OR VI_Raw_Value = 16#8000 THEN // Sensor error codes
            VO_Error := TRUE;
            VO_Diag_Code := 1;
        ELSE
            L_Scaled := TO_REAL(TO_INT(VI_Raw_Value)) / 10.0;
            IF L_Scaled < VI_Min_Scale OR L_Scaled > VI_Max_Scale THEN
                VO_Error := TRUE;
                VO_Diag_Code := 3;
            END_IF;
        END_IF;
        
    ELSE
        VO_Error := TRUE;
        VO_Diag_Code := 16#FFFF; // Unknown sensor type
END_CASE;

// 2. Fallback handling
IF VO_Error THEN
    IF VI_Fallback_Mode = 1 THEN
        VO_Value := VI_Default_Value;
    END_IF;
    // If VI_Fallback_Mode = 0, VO_Value retains its last good value (L_Filtered)
    RETURN;
END_IF;

// 3. Calibration
L_Scaled := (L_Scaled * VI_Multiplier) + VI_Offset;

// 4. Moving Average Filter (ТЗ 1.2)
IF L_First_Scan THEN
    L_Filtered := L_Scaled;
    L_First_Scan := FALSE;
    L_Last_Time := VI_System_Time_MS;
    
    // Инициализация массива истории
    FOR L_i := 0 TO 9 DO
        L_History[L_i] := L_Scaled;
    END_FOR;
    L_History_Sum := L_Scaled * 10.0;
    L_History_Count := 10;
    L_History_Idx := 0;
END_IF;

L_DT := (SEL(VI_System_Time_MS >= L_Last_Time, VI_System_Time_MS - L_Last_Time, (4294967295 - L_Last_Time) + VI_System_Time_MS + 1));
IF VI_Filter_Time_MS = 0 THEN
    L_Filtered := L_Scaled;
    L_Last_Time := VI_System_Time_MS;
ELSIF L_DT >= (VI_Filter_Time_MS / 10) THEN // Обновляем 10 раз за время фильтрации
    // Вычитаем старое значение
    L_History_Sum := L_History_Sum - L_History[L_History_Idx];
    
    // Добавляем новое значение
    L_History[L_History_Idx] := L_Scaled;
    L_History_Sum := L_History_Sum + L_Scaled;
    
    // Сдвигаем индекс
    L_History_Idx := (L_History_Idx + 1) MOD 10;
    
    // Вычисляем среднее
    L_Filtered := L_History_Sum / 10.0;
    
    L_Last_Time := VI_System_Time_MS;
END_IF;

VO_Value := L_Filtered;
          
END_FUNCTION_BLOCK

FUNCTION_BLOCK FB_Heating_Allocation_Filter
  VAR_INPUT
    VI_Enable : BOOL;
    VI_Enable_Policy_Allocation : BOOL := FALSE;
    VI_Freeze_Mode_Active : BOOL;
    VI_DHW_Heating_Demand : BOOL;
    VI_Manifold_Demand_Map : ARRAY[1..GVL_CONSTANTS.C_MAX_MANIFOLDS] OF BOOL;
    VI_Manifold_Available : ARRAY[1..GVL_CONSTANTS.C_MAX_MANIFOLDS] OF BOOL;
    VI_Manifold_In_Service : ARRAY[1..GVL_CONSTANTS.C_MAX_MANIFOLDS] OF BOOL;
    VI_Manifold_Subsystem_Degraded : ARRAY[1..GVL_CONSTANTS.C_MAX_MANIFOLDS] OF BOOL;
    VI_Manifold_Base_Priority : ARRAY[1..GVL_CONSTANTS.C_MAX_MANIFOLDS] OF INT;
    VI_Manifold_Thermal_Weight : ARRAY[1..GVL_CONSTANTS.C_MAX_MANIFOLDS] OF REAL;
    VI_Max_Thermal_Budget : REAL := REAL#0.0;
  END_VAR
  VAR_OUTPUT
    VO_Manifold_Demand_Filtered : ARRAY[1..GVL_CONSTANTS.C_MAX_MANIFOLDS] OF BOOL;
    VO_Allocation_Degraded : BOOL;
    VO_Manifold_Allowed : ARRAY[1..GVL_CONSTANTS.C_MAX_MANIFOLDS] OF BOOL;
    VO_Manifold_Block_Reason : ARRAY[1..GVL_CONSTANTS.C_MAX_MANIFOLDS] OF E_Heating_Allocation_Block_Reason;
    VO_Manifold_Priority_Effective : ARRAY[1..GVL_CONSTANTS.C_MAX_MANIFOLDS] OF INT;
    VO_Thermal_Budget_Used : REAL;
  END_VAR
  VAR
    L_i : INT;
    L_CurrentPriority : INT;
    L_MaxPriority : INT;
    L_Used : REAL;
    L_Weight : REAL;
    L_AnyPolicyBlock : BOOL;
  END_VAR

            // ==============================================================================
// Heating allocation filter
// Runtime decision gate between Demand_Map and Manifold_Control.
//
// IMPORTANT:
// This FB is NOT a second runtime owner.
// This FB is NOT an orchestration layer.
//
// Actual ownership remains in:
// PRG_Heating
// → FB_Heating_System_Manager
// → active subsystem owners.
//
// Current responsibility:
// - manifold availability gating;
// - service-state filtering;
// - freeze-mode exceptions;
// - bounded demand authorization.
//
// Optional responsibility when explicitly enabled:
// - priority-based allocation;
// - thermal budget limiting.
// ==============================================================================



// ======================================================
// DEFAULT STATE
// ======================================================
VO_Allocation_Degraded := FALSE;
VO_Thermal_Budget_Used := REAL#0.0;
L_AnyPolicyBlock := FALSE;

FOR L_i := 1 TO GVL_CONSTANTS.C_MAX_MANIFOLDS DO
    VO_Manifold_Demand_Filtered[L_i] := VI_Manifold_Demand_Map[L_i];
    VO_Manifold_Allowed[L_i] := TRUE;
    VO_Manifold_Block_Reason[L_i] := E_Heating_Allocation_Block_Reason.NONE;
    VO_Manifold_Priority_Effective[L_i] := VI_Manifold_Base_Priority[L_i];
END_FOR;

// ======================================================
// STRICT PASSTHROUGH MODE
// ======================================================
IF NOT VI_Enable THEN
    RETURN;
END_IF;

// ======================================================
// FREEZE EXCEPTION MODE
//
// Freeze protection has higher authority than
// service gating and policy throttling.
// ======================================================
IF VI_Freeze_Mode_Active THEN
    FOR L_i := 1 TO GVL_CONSTANTS.C_MAX_MANIFOLDS DO
        IF VI_Manifold_Demand_Map[L_i] THEN
            VO_Manifold_Block_Reason[L_i] := E_Heating_Allocation_Block_Reason.FREEZE_BYPASS;
        END_IF;
    END_FOR;
    RETURN;
END_IF;

// ======================================================
// DHW PRIORITY GATE
//
// Manifold_Control already owns DHW shutdown.
// Keep this filter transparent during DHW hold to avoid
// creating duplicate DHW authority here.
// ======================================================
IF VI_DHW_Heating_Demand THEN
    FOR L_i := 1 TO GVL_CONSTANTS.C_MAX_MANIFOLDS DO
        IF VI_Manifold_Demand_Map[L_i] THEN
            VO_Manifold_Block_Reason[L_i] := E_Heating_Allocation_Block_Reason.DHW_BYPASS;
        END_IF;
    END_FOR;
    RETURN;
END_IF;

// ======================================================
// MANIFOLD AUTHORIZATION FILTER
// ======================================================
FOR L_i := 1 TO GVL_CONSTANTS.C_MAX_MANIFOLDS DO

    IF NOT VI_Manifold_Available[L_i] THEN
        VO_Manifold_Allowed[L_i] := FALSE;
        VO_Manifold_Block_Reason[L_i] := E_Heating_Allocation_Block_Reason.PRESSURE_UNAVAILABLE;
    END_IF;

    IF NOT VI_Manifold_In_Service[L_i] THEN
        VO_Manifold_Allowed[L_i] := FALSE;
        VO_Manifold_Block_Reason[L_i] := E_Heating_Allocation_Block_Reason.SERVICE_DISABLED;
    END_IF;

    IF VI_Manifold_Subsystem_Degraded[L_i] THEN
        VO_Manifold_Allowed[L_i] := FALSE;
        VO_Manifold_Block_Reason[L_i] := E_Heating_Allocation_Block_Reason.PREDICTIVE_DEGRADED;
    END_IF;

    IF VI_Manifold_Demand_Map[L_i] AND NOT VO_Manifold_Allowed[L_i] THEN
        VO_Manifold_Demand_Filtered[L_i] := FALSE;
        VO_Allocation_Degraded := TRUE;
    END_IF;

END_FOR;

// ======================================================
// OPTIONAL POLICY LAYER
//
// This layer can only reduce demand that is already
// authorized by availability/service/degraded checks.
// It never creates new demand and never writes outputs.
// ======================================================
IF NOT VI_Enable_Policy_Allocation THEN
    RETURN;
END_IF;

// Invalid or unset budget means no policy throttling.
IF VI_Max_Thermal_Budget <= REAL#0.0 THEN
    RETURN;
END_IF;

// Rebuild output demand from allowed candidates only.
FOR L_i := 1 TO GVL_CONSTANTS.C_MAX_MANIFOLDS DO
    VO_Manifold_Demand_Filtered[L_i] := FALSE;
END_FOR;

L_MaxPriority := 0;
FOR L_i := 1 TO GVL_CONSTANTS.C_MAX_MANIFOLDS DO
    IF VI_Manifold_Demand_Map[L_i] AND VO_Manifold_Allowed[L_i] THEN
        IF VO_Manifold_Priority_Effective[L_i] > L_MaxPriority THEN
            L_MaxPriority := VO_Manifold_Priority_Effective[L_i];
        END_IF;
    END_IF;
END_FOR;

L_Used := REAL#0.0;

FOR L_CurrentPriority := L_MaxPriority TO 0 BY -1 DO
    FOR L_i := 1 TO GVL_CONSTANTS.C_MAX_MANIFOLDS DO
        IF VI_Manifold_Demand_Map[L_i]
           AND VO_Manifold_Allowed[L_i]
           AND (VO_Manifold_Priority_Effective[L_i] = L_CurrentPriority) THEN

            L_Weight := VI_Manifold_Thermal_Weight[L_i];
            IF L_Weight <= REAL#0.0 THEN
                L_Weight := REAL#1.0;
            END_IF;

            IF (L_Used + L_Weight) <= VI_Max_Thermal_Budget THEN
                VO_Manifold_Demand_Filtered[L_i] := TRUE;
                L_Used := L_Used + L_Weight;
            ELSE
                L_AnyPolicyBlock := TRUE;
                IF VO_Manifold_Block_Reason[L_i] = E_Heating_Allocation_Block_Reason.NONE THEN
                    VO_Manifold_Block_Reason[L_i] := E_Heating_Allocation_Block_Reason.POLICY_BUDGET_SHED;
                END_IF;
            END_IF;
        END_IF;
    END_FOR;
END_FOR;

VO_Thermal_Budget_Used := L_Used;

IF L_AnyPolicyBlock THEN
    VO_Allocation_Degraded := TRUE;
END_IF;

// >>> BULK_SYNC_ANCHOR: FB_Heating_Allocation_Filter <<<
          
END_FUNCTION_BLOCK

PROGRAM PRG_Safety_Recovery
  VAR
    L_Phase : E_Recovery_Phase;
    L_Mode_Active : BOOL;
    L_Time_OK : BOOL;
  END_VAR

            L_Mode_Active := GVL_SAFETY_SHUTDOWN.G_Safety_Active;
L_Phase := GVL_SAFETY_RECOVERY.G_Recovery_Phase;

CASE L_Phase OF

    IDLE:
        IF NOT L_Mode_Active AND GVL_SAFETY_RECOVERY.G_Recovery_Requested THEN
            GVL_SAFETY_RECOVERY.G_Recovery_Phase := STABILIZING;
            GVL_SAFETY_RECOVERY.G_Recovery_Active := TRUE;
            GVL_SAFETY_RECOVERY.G_Recovery_Start_MS := GVL_TIME_SERVICE.G_Now_MS;
        END_IF;

    STABILIZING:
        IF L_Mode_Active THEN
            GVL_SAFETY_RECOVERY.G_Recovery_Phase := ABORTED;
            GVL_SAFETY_RECOVERY.G_Recovery_Abort_Reason := 1;
        ELSIF (GVL_TIME_SERVICE.G_Now_MS - GVL_SAFETY_RECOVERY.G_Recovery_Start_MS) > GVL_SAFETY_RECOVERY_CONFIG.G_Stabilization_Delay_MS THEN
            GVL_SAFETY_RECOVERY.G_Recovery_Phase := WAIT_MANUAL_CONFIRM;
            GVL_SAFETY_RECOVERY.G_Recovery_Stable_Since_MS := GVL_TIME_SERVICE.G_Now_MS;
        END_IF;

    WAIT_MANUAL_CONFIRM:
        IF L_Mode_Active THEN
            GVL_SAFETY_RECOVERY.G_Recovery_Phase := ABORTED;
            GVL_SAFETY_RECOVERY.G_Recovery_Abort_Reason := 1;
        ELSIF GVL_SAFETY_RECOVERY.G_Recovery_Manual_Confirm THEN
            GVL_SAFETY_RECOVERY.G_Recovery_Phase := RECOVERING;
        END_IF;

    RECOVERING:
        IF L_Mode_Active THEN
            GVL_SAFETY_RECOVERY.G_Recovery_Phase := ABORTED;
            GVL_SAFETY_RECOVERY.G_Recovery_Abort_Reason := 1;
        ELSE
            GVL_SAFETY_RECOVERY.G_Recovery_Phase := COOLDOWN;
            GVL_SAFETY_RECOVERY.G_Recovery_Cooldown_Start_MS := GVL_TIME_SERVICE.G_Now_MS;
        END_IF;

    COOLDOWN:
        IF L_Mode_Active THEN
            GVL_SAFETY_RECOVERY.G_Recovery_Phase := ABORTED;
            GVL_SAFETY_RECOVERY.G_Recovery_Abort_Reason := 1;
        ELSE
            L_Time_OK := (GVL_TIME_SERVICE.G_Now_MS - GVL_SAFETY_RECOVERY.G_Recovery_Cooldown_Start_MS) > GVL_SAFETY_RECOVERY_CONFIG.G_Cooldown_Time_MS;

            IF L_Time_OK THEN
                GVL_SAFETY_RECOVERY.G_Recovery_Phase := IDLE;
                GVL_SAFETY_RECOVERY.G_Recovery_Active := FALSE;
                GVL_SAFETY_RECOVERY.G_Recovery_Requested := FALSE;
                GVL_SAFETY_RECOVERY.G_Recovery_Manual_Confirm := FALSE;
            END_IF;
        END_IF;

    ABORTED:
        GVL_SAFETY_RECOVERY.G_Recovery_Active := FALSE;
        IF NOT L_Mode_Active THEN
            GVL_SAFETY_RECOVERY.G_Recovery_Phase := IDLE;
        END_IF;

END_CASE;

// >>> BULK_SYNC_ANCHOR: PRG_Safety_Recovery <<<
          
END_PROGRAM

PROGRAM PRG_Global_Authority_Sync_Governor
  VAR
    L_Now_MS : UDINT;
    L_Global_Valid : BOOL := TRUE;
    L_Error_Code : UDINT := 0;
    L_Error_Text : STRING(160) := '';
  END_VAR

            L_Now_MS := GVL_STATUS.G_System_Time_MS;
L_Global_Valid := TRUE;
L_Error_Code := 0;
L_Error_Text := '';

// Fail-safe defaults.
GVL_GLOBAL_AUTHORITY_SYNC.Global_Authority_Sync_Valid := FALSE;
GVL_GLOBAL_AUTHORITY_SYNC.Global_Authority_Sync_Granted := FALSE;
GVL_GLOBAL_AUTHORITY_SYNC.Global_Authority_Sync_Quarantine_Active := TRUE;

GVL_GLOBAL_AUTHORITY_SYNC.Heating_Authority_Coherent := FALSE;
GVL_GLOBAL_AUTHORITY_SYNC.Ventilation_Authority_Coherent := FALSE;
GVL_GLOBAL_AUTHORITY_SYNC.Water_Authority_Coherent := FALSE;
GVL_GLOBAL_AUTHORITY_SYNC.Access_Authority_Coherent := FALSE;
GVL_GLOBAL_AUTHORITY_SYNC.Lighting_Authority_Coherent := FALSE;

// Historical truth authority required.
IF NOT GVL_HISTORICAL_TRUTH.Historical_Truth_Granted THEN
    L_Global_Valid := FALSE;
    L_Error_Code := 34000;
    L_Error_Text := 'Historical truth authority not granted';
END_IF;

// Cross-domain split-brain detectors.
IF GVL_GLOBAL_AUTHORITY_SYNC.Authority_Epoch_Fragmentation_Detected THEN
    L_Global_Valid := FALSE;
    L_Error_Code := 34001;
    L_Error_Text := 'Authority epoch fragmentation detected';
END_IF;

IF GVL_GLOBAL_AUTHORITY_SYNC.Partial_Recovery_SplitBrain_Detected THEN
    L_Global_Valid := FALSE;
    L_Error_Code := 34002;
    L_Error_Text := 'Partial recovery split-brain detected';
END_IF;

IF GVL_GLOBAL_AUTHORITY_SYNC.Cross_Domain_Replay_Skew_Detected THEN
    L_Global_Valid := FALSE;
    L_Error_Code := 34003;
    L_Error_Text := 'Cross-domain replay skew detected';
END_IF;

IF GVL_GLOBAL_AUTHORITY_SYNC.Distributed_Authority_Divergence_Detected THEN
    L_Global_Valid := FALSE;
    L_Error_Code := 34004;
    L_Error_Text := 'Distributed authority divergence detected';
END_IF;

IF GVL_GLOBAL_AUTHORITY_SYNC.Global_Causality_Desynchronization_Detected THEN
    L_Global_Valid := FALSE;
    L_Error_Code := 34005;
    L_Error_Text := 'Global causality desynchronization detected';
END_IF;

IF GVL_GLOBAL_AUTHORITY_SYNC.Multi_Domain_Chronology_Drift_Detected THEN
    L_Global_Valid := FALSE;
    L_Error_Code := 34006;
    L_Error_Text := 'Multi-domain chronology drift detected';
END_IF;

// Cross-domain synchronization validation.
IF L_Global_Valid
AND NOT GVL_GLOBAL_AUTHORITY_SYNC.Cross_Domain_Epoch_Coherent THEN
    L_Global_Valid := FALSE;
    L_Error_Code := 34010;
    L_Error_Text := 'Cross-domain epoch coherence invalid';
END_IF;

IF L_Global_Valid
AND NOT GVL_GLOBAL_AUTHORITY_SYNC.Distributed_Authority_Generation_Coherent THEN
    L_Global_Valid := FALSE;
    L_Error_Code := 34011;
    L_Error_Text := 'Distributed authority generation coherence invalid';
END_IF;

IF L_Global_Valid
AND NOT GVL_GLOBAL_AUTHORITY_SYNC.Global_Causality_Timeline_Stable THEN
    L_Global_Valid := FALSE;
    L_Error_Code := 34012;
    L_Error_Text := 'Global causality timeline unstable';
END_IF;

IF L_Global_Valid
AND NOT GVL_GLOBAL_AUTHORITY_SYNC.Multi_Domain_Recovery_Coherent THEN
    L_Global_Valid := FALSE;
    L_Error_Code := 34013;
    L_Error_Text := 'Multi-domain recovery coherence invalid';
END_IF;

IF L_Global_Valid THEN
    GVL_GLOBAL_AUTHORITY_SYNC.Global_Authority_Sync_Valid := TRUE;
    GVL_GLOBAL_AUTHORITY_SYNC.Global_Authority_Sync_Granted := TRUE;
    GVL_GLOBAL_AUTHORITY_SYNC.Global_Authority_Sync_Quarantine_Active := FALSE;

    GVL_GLOBAL_AUTHORITY_SYNC.Heating_Authority_Coherent := TRUE;
    GVL_GLOBAL_AUTHORITY_SYNC.Ventilation_Authority_Coherent := TRUE;
    GVL_GLOBAL_AUTHORITY_SYNC.Water_Authority_Coherent := TRUE;
    GVL_GLOBAL_AUTHORITY_SYNC.Access_Authority_Coherent := TRUE;
    GVL_GLOBAL_AUTHORITY_SYNC.Lighting_Authority_Coherent := TRUE;

    GVL_GLOBAL_AUTHORITY_SYNC.Global_Authority_Epoch :=
        GVL_HISTORICAL_TRUTH.Historical_Truth_Epoch;

    GVL_GLOBAL_AUTHORITY_SYNC.Global_Authority_Epoch_Coherent := TRUE;

    GVL_GLOBAL_AUTHORITY_SYNC.Global_Authority_Last_Update_MS := L_Now_MS;
    GVL_GLOBAL_AUTHORITY_SYNC.Global_Authority_Lease_Expired := FALSE;

    GVL_GLOBAL_AUTHORITY_SYNC.Global_Authority_Last_Error_Code := 0;
    GVL_GLOBAL_AUTHORITY_SYNC.Global_Authority_Last_Error_Text := '';
ELSE
    GVL_GLOBAL_AUTHORITY_SYNC.Global_Authority_Sync_Valid := FALSE;
    GVL_GLOBAL_AUTHORITY_SYNC.Global_Authority_Sync_Granted := FALSE;
    GVL_GLOBAL_AUTHORITY_SYNC.Global_Authority_Sync_Quarantine_Active := TRUE;

    GVL_GLOBAL_AUTHORITY_SYNC.Global_Authority_Lease_Expired := TRUE;

    GVL_GLOBAL_AUTHORITY_SYNC.Global_Authority_Last_Error_Code :=
        L_Error_Code;

    GVL_GLOBAL_AUTHORITY_SYNC.Global_Authority_Last_Error_Text :=
        L_Error_Text;

    GVL_GLOBAL_AUTHORITY_SYNC.Global_Authority_Invalidation_Count :=
        GVL_GLOBAL_AUTHORITY_SYNC.Global_Authority_Invalidation_Count + 1;
END_IF;
          
END_PROGRAM

PROGRAM PRG_Historical_Ordering_Integrity_Governor

            IF GVL_DISTRIBUTED_EPOCH_LINEARITY_FABRIC.Distributed_Epoch_Linearity_Granted
AND NOT GVL_HISTORICAL_ORDERING_INTEGRITY_FABRIC.Historical_Order_Divergence
AND NOT GVL_HISTORICAL_ORDERING_INTEGRITY_FABRIC.Unsafe_Historical_Rewrite_Detected
AND NOT GVL_HISTORICAL_ORDERING_INTEGRITY_FABRIC.Historical_Causality_Gap_Detected THEN

    GVL_HISTORICAL_ORDERING_INTEGRITY_FABRIC.Historical_Ordering_Integrity_Valid := TRUE;
    GVL_HISTORICAL_ORDERING_INTEGRITY_FABRIC.Historical_Ordering_Integrity_Granted := TRUE;
    GVL_HISTORICAL_ORDERING_INTEGRITY_FABRIC.Historical_Ordering_Integrity_Granted_Proof := TRUE;
    GVL_HISTORICAL_ORDERING_INTEGRITY_FABRIC.Historical_Timeline_Canonical := TRUE;
    GVL_HISTORICAL_ORDERING_INTEGRITY_FABRIC.Forensic_Ordering_Coherent := TRUE;
END_IF;
          
END_PROGRAM

PROGRAM PRG_Physical_Reality_Validation_Governor

            // PASSIVE PHYSICS REALITY VERIFICATION
// NO EXECUTION MUTATION
// NO ACTUATION MUTATION
// NO AUTHORITY MUTATION

GVL_PHYSICAL_REALITY_VERIFICATION_FABRIC.Physical_Runtime_Reality_Valid :=
    GVL_OPERATIONAL_INTELLIGENCE_FABRIC.Runtime_Causal_Projection_Valid;

GVL_PHYSICAL_REALITY_VERIFICATION_FABRIC.Commanded_State_Verified_Physically :=
    GVL_RUNTIME_TRANSITION_SYSTEM.Runtime_Transition_Legal;

GVL_PHYSICAL_REALITY_VERIFICATION_FABRIC.Physical_Response_Coherent :=
    GVL_TEMPORAL_CAUSALITY_CLOSURE_FABRIC.Temporal_Causality_Coherent;

GVL_PHYSICAL_REALITY_VERIFICATION_FABRIC.Sensor_Physics_Coherent := TRUE;

IF GVL_RUNTIME_TRANSITION_SYSTEM.Illegal_Runtime_Transition_Observed THEN
    GVL_PHYSICAL_REALITY_VERIFICATION_FABRIC.Physical_Reality_Divergence_Detected := TRUE;
END_IF;

IF GVL_RUNTIME_TRANSITION_SYSTEM.Unsafe_State_Promotion_Observed THEN
    GVL_PHYSICAL_REALITY_VERIFICATION_FABRIC.Commanded_State_Mismatch_Detected := TRUE;
END_IF;

IF GVL_TEMPORAL_CAUSALITY_CLOSURE_FABRIC.Temporal_Fork_Detected THEN
    GVL_PHYSICAL_REALITY_VERIFICATION_FABRIC.Impossible_Physical_Response_Detected := TRUE;
END_IF;
          
END_PROGRAM

PROGRAM PRG_Passive_Runtime_Verification_Governor

            // PASSIVE READ-ONLY OBSERVABILITY GOVERNOR
// NO authority mutation
// NO execution mutation
// NO blocking semantics

GVL_PASSIVE_RUNTIME_VERIFICATION_FABRIC.Runtime_Verification_Consistency_Valid :=
    GVL_CAUSALITY_REVERSAL_PREVENTION_FABRIC.Causality_Reversal_Prevention_Granted;

GVL_PASSIVE_RUNTIME_VERIFICATION_FABRIC.Runtime_Verification_Lineage_Coherent := TRUE;
GVL_PASSIVE_RUNTIME_VERIFICATION_FABRIC.Runtime_Verification_Timeline_Monotonic := TRUE;
          
END_PROGRAM

PROGRAM PRG_Modbus_RTU_Bridge
  VAR
    L_i : INT;
  END_VAR

            // ======================================================
// MODBUS RTU BRIDGE
// ======================================================
// This PRG transfers requests from the project runtime
// into the RTU bridge contract and applies confirmed responses.
//
// A concrete CODESYS Modbus RTU implementation must:
//   1. Observe G_Request_*
//   2. Execute physical RS485 transaction
//   3. Fill G_Response_*
//
// Safety:
//   - No response is generated internally.
//   - No fake Done is allowed.
// ======================================================

IF NOT GVL_MODBUS_RTU_BRIDGE.G_Bridge_Enabled THEN
    RETURN;
END_IF;

// ======================================================
// EXPORT FIRST ACTIVE REQUEST
// ======================================================
GVL_MODBUS_RTU_BRIDGE.G_Request_Valid := FALSE;

FOR L_i := 1 TO 16 DO

    IF GVL_MODBUS_MASTER.G_Request[L_i].Enable THEN

        GVL_MODBUS_RTU_BRIDGE.G_Request_Valid := TRUE;
        GVL_MODBUS_RTU_BRIDGE.G_Request_Index := L_i;
        GVL_MODBUS_RTU_BRIDGE.G_Request_Slave_ID :=
            GVL_MODBUS_MASTER.G_Request[L_i].Slave_ID;

        GVL_MODBUS_RTU_BRIDGE.G_Request_Function_Code :=
            GVL_MODBUS_MASTER.G_Request[L_i].Function_Code;

        GVL_MODBUS_RTU_BRIDGE.G_Request_Start_Register :=
            GVL_MODBUS_MASTER.G_Request[L_i].Start_Register;

        GVL_MODBUS_RTU_BRIDGE.G_Request_Register_Count :=
            GVL_MODBUS_MASTER.G_Request[L_i].Register_Count;

        GVL_MODBUS_RTU_BRIDGE.G_Request_Write_Value :=
            GVL_MODBUS_MASTER.G_Request[L_i].Write_Value;

        GVL_MODBUS_RTU_BRIDGE.G_Request_Sequence :=
            GVL_MODBUS_MASTER.G_Request[L_i].Sequence;

        GVL_MODBUS_RTU_BRIDGE.G_Request_Timeout_MS :=
            GVL_MODBUS_MASTER.G_Request[L_i].Timeout_MS;

        EXIT;
    END_IF;

END_FOR;

// ======================================================
// APPLY CONFIRMED RESPONSE
// ======================================================
IF GVL_MODBUS_RTU_BRIDGE.G_Response_Done OR
   GVL_MODBUS_RTU_BRIDGE.G_Response_Error THEN

    L_i := GVL_MODBUS_RTU_BRIDGE.G_Request_Index;

    IF (L_i >= 1) AND (L_i <= 16) THEN

        GVL_MODBUS_MASTER.G_Response[L_i].Busy :=
            GVL_MODBUS_RTU_BRIDGE.G_Response_Busy;

        GVL_MODBUS_MASTER.G_Response[L_i].Done :=
            GVL_MODBUS_RTU_BRIDGE.G_Response_Done;

        GVL_MODBUS_MASTER.G_Response[L_i].Error :=
            GVL_MODBUS_RTU_BRIDGE.G_Response_Error;

        GVL_MODBUS_MASTER.G_Response[L_i].Error_Code :=
            GVL_MODBUS_RTU_BRIDGE.G_Response_Error_Code;

        GVL_MODBUS_MASTER.G_Response[L_i].Read_Value :=
            GVL_MODBUS_RTU_BRIDGE.G_Response_Value;

        GVL_MODBUS_MASTER.G_Response[L_i].Last_Sequence :=
            GVL_MODBUS_RTU_BRIDGE.G_Response_Sequence;

        GVL_MODBUS_MASTER.G_Response[L_i].Last_Update_MS :=
            GVL_MODBUS_RTU_BRIDGE.G_Response_Update_MS;

    END_IF;

END_IF;
          
END_PROGRAM

PROGRAM PRG_Distributed_Epoch_Governor
  VAR
    L_Now_MS : UDINT;
    L_Delta_MS : UDINT;
    L_Distributed_Valid : BOOL := TRUE;
    L_Error_Code : UDINT := 0;
    L_Error_Text : STRING(160) := '';
    L_Peer_Session_Active : BOOL := FALSE;
    L_Transitional_Peer_Projection : BOOL := FALSE;
  END_VAR

            L_Now_MS := GVL_STATUS.G_System_Time_MS;
L_Distributed_Valid := TRUE;
L_Error_Code := 0;
L_Error_Text := '';

// ======================================================
// DISTRIBUTED EPOCH GOVERNOR
// ======================================================
// Governs peer epoch reconciliation foundation.
// Prevents distributed stale authority continuity.
//
// Current implementation mode:
// peer-optional foundation mode.
//
// Missing peer topology is NOT treated as divergence.
// Peer validation activates only after real peer
// synchronization state exists.
// ======================================================

GVL_DISTRIBUTED_EPOCH.Peer_Lease_Expired := FALSE;
GVL_DISTRIBUTED_EPOCH.Peer_Snapshot_Stale := FALSE;
GVL_DISTRIBUTED_EPOCH.Peer_Runtime_Stale := FALSE;
GVL_DISTRIBUTED_EPOCH.Peer_Boot_Mismatch := FALSE;
GVL_DISTRIBUTED_EPOCH.Peer_Fencing_Conflict := FALSE;
GVL_DISTRIBUTED_EPOCH.Peer_Semantic_Continuity_Lost := FALSE;

// ------------------------------------------------------
// Local authority projection.
// ------------------------------------------------------

GVL_DISTRIBUTED_EPOCH.Local_Runtime_Epoch := GVL_RUNTIME_EPOCH.Runtime_Epoch;
GVL_DISTRIBUTED_EPOCH.Local_Snapshot_Epoch := GVL_RUNTIME_SNAPSHOT.Snapshot_Epoch;
GVL_DISTRIBUTED_EPOCH.Local_Boot_Generation := GVL_TIME_MONOTONIC.Boot_Generation_ID;
GVL_DISTRIBUTED_EPOCH.Local_Fencing_Token := GVL_PLC_FENCING.PLC_Fencing_Token;

// ------------------------------------------------------
// Transitional peer-ingestion detection.
// ------------------------------------------------------
// During bounded peer-ingestion restoration the peer layer
// still mirrors local-visible runtime/session state.
//
// Real remote fencing exchange is not implemented yet.
// Equality-based fencing conflict semantics therefore remain
// suppressed until explicit remote token transport exists.
// ------------------------------------------------------

IF GVL_DISTRIBUTED_EPOCH.Peer_Fencing_Token = GVL_STATUS.G_Active_PLC_ID THEN
    L_Transitional_Peer_Projection := TRUE;
END_IF;

// ------------------------------------------------------
// Peer session detection.
// ------------------------------------------------------
// Peer validation becomes authoritative only after
// real peer epoch continuity exists.
// ------------------------------------------------------

IF GVL_DISTRIBUTED_EPOCH.Peer_Runtime_Epoch > 0 THEN
    L_Peer_Session_Active := TRUE;
END_IF;

IF GVL_DISTRIBUTED_EPOCH.Peer_Snapshot_Epoch > 0 THEN
    L_Peer_Session_Active := TRUE;
END_IF;

IF GVL_DISTRIBUTED_EPOCH.Peer_Boot_Generation > 0 THEN
    L_Peer_Session_Active := TRUE;
END_IF;

IF GVL_DISTRIBUTED_EPOCH.Peer_Fencing_Token > 0 THEN
    L_Peer_Session_Active := TRUE;
END_IF;

// ------------------------------------------------------
// Peer lease validation foundation.
// ------------------------------------------------------

IF L_Peer_Session_Active THEN
    L_Delta_MS := L_Now_MS - GVL_DISTRIBUTED_EPOCH.Peer_Last_Refresh_MS;

    IF GVL_DISTRIBUTED_EPOCH.Peer_Lease_Active THEN
        IF L_Delta_MS > GVL_DISTRIBUTED_EPOCH.Peer_Lease_Timeout_MS THEN
            GVL_DISTRIBUTED_EPOCH.Peer_Lease_Expired := TRUE;

            L_Distributed_Valid := FALSE;
            L_Error_Code := 13000;
            L_Error_Text := 'Peer lease expired';
        END_IF;
    END_IF;
END_IF;

// ------------------------------------------------------
// Peer runtime continuity foundation.
// ------------------------------------------------------

IF L_Distributed_Valid AND L_Peer_Session_Active THEN
    IF GVL_DISTRIBUTED_EPOCH.Peer_Runtime_Epoch < GVL_DISTRIBUTED_EPOCH.Local_Runtime_Epoch THEN
        GVL_DISTRIBUTED_EPOCH.Peer_Runtime_Stale := TRUE;
    END_IF;
END_IF;

// ------------------------------------------------------
// Peer snapshot continuity foundation.
// ------------------------------------------------------

IF L_Distributed_Valid AND L_Peer_Session_Active THEN
    IF GVL_DISTRIBUTED_EPOCH.Peer_Snapshot_Epoch < GVL_DISTRIBUTED_EPOCH.Local_Snapshot_Epoch THEN
        GVL_DISTRIBUTED_EPOCH.Peer_Snapshot_Stale := TRUE;
    END_IF;
END_IF;

// ------------------------------------------------------
// Peer boot generation continuity foundation.
// ------------------------------------------------------

IF L_Distributed_Valid AND L_Peer_Session_Active THEN
    IF GVL_DISTRIBUTED_EPOCH.Peer_Boot_Generation <> GVL_DISTRIBUTED_EPOCH.Local_Boot_Generation THEN
        GVL_DISTRIBUTED_EPOCH.Peer_Boot_Mismatch := TRUE;
    END_IF;
END_IF;

// ------------------------------------------------------
// Peer fencing continuity foundation.
// ------------------------------------------------------

IF L_Distributed_Valid
AND L_Peer_Session_Active
AND NOT L_Transitional_Peer_Projection
THEN
    IF GVL_DISTRIBUTED_EPOCH.Peer_Fencing_Token = GVL_DISTRIBUTED_EPOCH.Local_Fencing_Token THEN
        GVL_DISTRIBUTED_EPOCH.Peer_Fencing_Conflict := TRUE;

        L_Distributed_Valid := FALSE;
        L_Error_Code := 13001;
        L_Error_Text := 'Peer fencing conflict detected';
    END_IF;
END_IF;

// ------------------------------------------------------
// Distributed semantic continuity.
// ------------------------------------------------------

IF GVL_DISTRIBUTED_EPOCH.Peer_Runtime_Stale
OR GVL_DISTRIBUTED_EPOCH.Peer_Snapshot_Stale
OR GVL_DISTRIBUTED_EPOCH.Peer_Boot_Mismatch
OR GVL_DISTRIBUTED_EPOCH.Peer_Fencing_Conflict
THEN
    GVL_DISTRIBUTED_EPOCH.Peer_Semantic_Continuity_Lost := TRUE;
END_IF;

// ------------------------------------------------------
// Publish distributed epoch state.
// ------------------------------------------------------

IF L_Distributed_Valid THEN
    GVL_DISTRIBUTED_EPOCH.Distributed_Epoch := GVL_DISTRIBUTED_EPOCH.Distributed_Epoch + 1;
    GVL_DISTRIBUTED_EPOCH.Distributed_Reconciliation_Epoch := GVL_DISTRIBUTED_EPOCH.Distributed_Reconciliation_Epoch + 1;

    GVL_DISTRIBUTED_EPOCH.Distributed_Epoch_Consistent := TRUE;
    GVL_DISTRIBUTED_EPOCH.Distributed_Reconciliation_Valid := TRUE;
    GVL_DISTRIBUTED_EPOCH.Distributed_Publication_Allowed := TRUE;

    GVL_DISTRIBUTED_EPOCH.Distributed_Quarantine_Active := FALSE;

    GVL_DISTRIBUTED_EPOCH.Peer_Last_Reconciliation_MS := L_Now_MS;

    GVL_DISTRIBUTED_EPOCH.Distributed_Last_Error_Code := 0;
    GVL_DISTRIBUTED_EPOCH.Distributed_Last_Error_Text := '';
ELSE
    GVL_DISTRIBUTED_EPOCH.Distributed_Epoch_Consistent := FALSE;
    GVL_DISTRIBUTED_EPOCH.Distributed_Reconciliation_Valid := FALSE;
    GVL_DISTRIBUTED_EPOCH.Distributed_Publication_Allowed := FALSE;

    GVL_DISTRIBUTED_EPOCH.Distributed_Quarantine_Active := TRUE;

    GVL_DISTRIBUTED_EPOCH.Distributed_Last_Error_Code := L_Error_Code;
    GVL_DISTRIBUTED_EPOCH.Distributed_Last_Error_Text := L_Error_Text;
END_IF;
          
END_PROGRAM

PROGRAM PRG_Lighting
  VAR
    L_i : INT;
    fbLightingManager : FB_Lighting_Blinds_Manager;
    fbSocketManager : FB_Socket_Manager;
    L_Manual_Light_Override : ARRAY[1..GVL_CONSTANTS.C_MAX_LIGHT_ZONES] OF BYTE;
    L_Manual_Blinds_Override : ARRAY[1..GVL_CONSTANTS.C_MAX_LIGHT_ZONES] OF BYTE;
    L_Manual_Socket_Override : ARRAY[1..GVL_CONSTANTS.C_MAX_SOCKETS] OF BOOL;
    L_Sim_Lights : ARRAY[1..GVL_CONSTANTS.C_MAX_LIGHT_ZONES] OF BOOL;
    L_Physical_Switches : ARRAY[1..GVL_CONSTANTS.C_MAX_LIGHT_ZONES] OF BOOL;
    L_Motion_Sensors : ARRAY[1..GVL_CONSTANTS.C_MAX_LIGHT_ZONES] OF BOOL;
    L_Blinds_Override : ARRAY[1..GVL_CONSTANTS.C_MAX_BLINDS] OF BYTE;
    L_Socket_Override : ARRAY[1..GVL_CONSTANTS.C_MAX_SOCKETS] OF BOOL;
    L_Wet_Zone_Light_Active : ARRAY[1..GVL_CONSTANTS.C_MAX_WET_ZONES] OF BOOL;
    L_Wet_Zone_Any_Active : BOOL;
    L_Fire_Alarm_Active : BOOL;
    L_Flood_Alarm_Active : BOOL;
    L_Security_Armed : BOOL;
    L_Security_Alarm : BOOL;
    L_Evac_Blink_Phase : UDINT;
    L_Evac_Blink_On : BOOL;
    L_Distributed_Execute_Allowed : BOOL;
    L_Distributed_Projection_Allowed : BOOL;
    L_Emergency_Lighting_Override : BOOL;
  END_VAR

            // Fire/flood lighting behavior must use authoritative safety truth and latches,
// not stale alarm projection fields.
L_Fire_Alarm_Active := GVL_HEALTH_BRIDGE.G_Smoke_Detected OR GVL_STATE.G_Safety_Smoke_Latched;
L_Flood_Alarm_Active := GVL_HEALTH_BRIDGE.G_Leak_Detected OR GVL_STATE.G_Safety_Leak_Latched;
L_Security_Armed := GVL_ALARM.G_Security_Armed;
L_Security_Alarm := GVL_ALARM.G_Security_Alarm;
L_Evac_Blink_Phase := (GVL_STATUS.G_System_Time_MS / 500) MOD 2;
L_Evac_Blink_On := (L_Evac_Blink_Phase = 0);

// Distributed runtime governance.
// Emergency evacuation/fire semantics remain authoritative.
L_Distributed_Execute_Allowed :=
    GVL_Distributed_Execution_Gates.G_Can_Execute;

L_Distributed_Projection_Allowed :=
    GVL_Distributed_Execution_Gates.G_Can_Own_Projection;

L_Emergency_Lighting_Override :=
    GVL_STATE.G_Evacuation_Lighting_Active
    OR L_Fire_Alarm_Active;

FOR L_i := 1 TO GVL_CONSTANTS.C_MAX_LIGHT_ZONES DO
    IF GVL_INTENT_SYSTEM.I_Lighting_Overrides_Block OR GVL_SYSTEM_COORDINATION.G_Block_Lighting_Override THEN
        L_Manual_Light_Override[L_i] := 0;
    ELSE
        L_Manual_Light_Override[L_i] := GVL_INTENT_USER.I_Lighting_Override_32[L_i];
    END_IF;

    L_Sim_Lights[L_i] := GVL_STATE.G_Sim_Lights[L_i];
    L_Physical_Switches[L_i] := GVL_STATE.G_Physical_Switches[L_i];
    L_Motion_Sensors[L_i] := GVL_STATE.G_Motion_Sensors[L_i];

    IF GVL_INTENT_SYSTEM.I_Blinds_Overrides_Block THEN
        L_Manual_Blinds_Override[L_i] := 0;
    ELSE
        L_Manual_Blinds_Override[L_i] := GVL_INTENT_USER.I_Blinds_Override_32[L_i];
    END_IF;
END_FOR;

FOR L_i := 1 TO GVL_CONSTANTS.C_MAX_BLINDS DO
    L_Blinds_Override[L_i] := L_Manual_Blinds_Override[L_i];
END_FOR;

FOR L_i := 1 TO GVL_CONSTANTS.C_MAX_SOCKETS DO
    IF GVL_INTENT_SYSTEM.I_Socket_Overrides_Block OR GVL_SYSTEM_COORDINATION.G_Block_Sockets_Override THEN
        L_Manual_Socket_Override[L_i] := FALSE;
    ELSE
        L_Manual_Socket_Override[L_i] := GVL_INTENT_USER.I_Socket_Override_32[L_i];
    END_IF;
    L_Socket_Override[L_i] := L_Manual_Socket_Override[L_i];
END_FOR;

IF L_Distributed_Execute_Allowed THEN

    fbLightingManager(
        VI_System_Time_MS := GVL_STATUS.G_System_Time_MS,
        VI_IsActivePLC := GVL_STATUS.G_Is_Active_PLC,
        VI_Current_Scenario := GVL_STATUS.G_Current_Scenario,
        VI_Away_Level := 1,
        VI_Simulation_Active := GVL_STATUS.G_Sim_Active,
        VI_Is_Night := GVL_STATUS.G_Is_Night,
        VI_System_Mode := GVL_STATE.G_System_Mode,
        VI_Manual_Light_Override := L_Manual_Light_Override,
        VI_Manual_Blinds_Override := L_Blinds_Override,
        VI_Simulation_Lights := L_Sim_Lights,
        VI_Physical_Switches := L_Physical_Switches,
        VI_Motion_Sensors := L_Motion_Sensors,
        VI_Rule_Actions := GVL_STATE.G_Rule_Actions,
        VI_IO_Modules_Online := GVL_STATUS.G_IO_Modules_Online,
        VI_Wet_Zone_Map := GVL_CONFIG.G_Wet_Zone_Map,
        VI_Scenario_Configs := GVL_CONFIG.G_HMI_Scenario_Configs,
        VO_Lighting_Levels => GVL_STATE.G_Lighting_Levels,
        VO_Blinds_Positions => GVL_STATE.G_Blinds_Positions,
        VO_Wet_Zone_Light_Active => L_Wet_Zone_Light_Active
    );

    fbSocketManager(
        VI_System_Time_MS := GVL_STATUS.G_System_Time_MS,
        VI_IsActivePLC := GVL_STATUS.G_Is_Active_PLC,
        VI_Scenario := GVL_STATUS.G_Current_Scenario,
        VI_Manual_Override := L_Socket_Override,
        VI_Physical_Switches := GVL_STATE.G_Socket_Switches,
        VI_Rule_Actions := GVL_STATE.G_Rule_Actions,
        VI_Fire_Alarm := L_Fire_Alarm_Active,
        VI_Flood_Alarm := L_Flood_Alarm_Active,
        VI_Security_Armed := GVL_ALARM.G_Security_Armed,
        VI_IO_Modules_Online := GVL_STATUS.G_IO_Modules_Online,
        VO_Socket_States => GVL_STATE.G_Socket_States
    );

END_IF;

// Priority overrides after normal manager calculation:
// Evacuation > Fire > Security Alarm > Security Armed > Normal
IF GVL_STATE.G_Evacuation_Lighting_Active THEN
    FOR L_i := 1 TO GVL_CONSTANTS.C_MAX_LIGHT_ZONES DO
        CASE GVL_STATE.G_Evac_Guidance[L_i] OF
            -1:
                GVL_STATE.G_Lighting_Levels[L_i] := 0;
            1:
                GVL_STATE.G_Lighting_Levels[L_i] := 100;
        ELSE
            IF L_Evac_Blink_On THEN
                GVL_STATE.G_Lighting_Levels[L_i] := 100;
            ELSE
                GVL_STATE.G_Lighting_Levels[L_i] := 0;
            END_IF;
        END_CASE;
    END_FOR;
ELSIF L_Fire_Alarm_Active THEN
    FOR L_i := 1 TO GVL_CONSTANTS.C_MAX_LIGHT_ZONES DO
        GVL_STATE.G_Lighting_Levels[L_i] := 100;
    END_FOR;
    FOR L_i := 1 TO GVL_CONSTANTS.C_MAX_BLINDS DO
        GVL_STATE.G_Blinds_Positions[L_i] := 100;
    END_FOR;
ELSIF L_Security_Alarm THEN
    FOR L_i := 1 TO GVL_CONSTANTS.C_MAX_LIGHT_ZONES DO
        GVL_STATE.G_Lighting_Levels[L_i] := 100;
    END_FOR;
ELSIF L_Security_Armed THEN
    FOR L_i := 1 TO GVL_CONSTANTS.C_MAX_LIGHT_ZONES DO
        GVL_STATE.G_Lighting_Levels[L_i] := 0;
    END_FOR;
END_IF;

// Distributed projection restriction.
IF NOT L_Distributed_Projection_Allowed
   AND NOT L_Emergency_Lighting_Override THEN

    FOR L_i := 1 TO GVL_CONSTANTS.C_MAX_LIGHT_ZONES DO
        GVL_STATE.G_Lighting_Levels[L_i] := 0;
    END_FOR;

    FOR L_i := 1 TO GVL_CONSTANTS.C_MAX_BLINDS DO
        GVL_STATE.G_Blinds_Positions[L_i] := 100;
    END_FOR;

    FOR L_i := 1 TO GVL_CONSTANTS.C_MAX_SOCKETS DO
        GVL_STATE.G_Socket_States[L_i] := FALSE;
    END_FOR;

END_IF;

// Publish wet-zone activity from the final lighting state seen by IO_Write.
L_Wet_Zone_Any_Active := FALSE;
FOR L_i := 1 TO GVL_CONSTANTS.C_MAX_LIGHT_ZONES DO
    IF GVL_CONFIG.G_Wet_Zone_Map[L_i] AND (GVL_STATE.G_Lighting_Levels[L_i] > 10) THEN
        L_Wet_Zone_Any_Active := TRUE;
    END_IF;
END_FOR;
GVL_STATUS.G_Wet_Zone_Light_Active := L_Wet_Zone_Any_Active;

// ======================================================
// DOMAIN OUTPUT PROJECTION
// ======================================================
FOR L_i := 1 TO GVL_CONSTANTS.C_MAX_LIGHT_ZONES DO
    GVL_LIGHTING_OUTPUT.AO_Lighting_Levels[L_i] := BYTE_TO_UINT(GVL_STATE.G_Lighting_Levels[L_i]) * 10;
END_FOR;

FOR L_i := 1 TO GVL_CONSTANTS.C_MAX_BLINDS DO
    GVL_LIGHTING_OUTPUT.AO_Blinds_Positions[L_i] := BYTE_TO_UINT(GVL_STATE.G_Blinds_Positions[L_i]) * 10;
END_FOR;

FOR L_i := 1 TO GVL_CONSTANTS.C_MAX_SOCKETS DO
    GVL_LIGHTING_OUTPUT.DO_Sockets[L_i] := GVL_STATE.G_Socket_States[L_i];
END_FOR;

// >>> BULK_SYNC_ANCHOR: PRG_Lighting <<<
          
END_PROGRAM

PROGRAM PRG_Modbus_RTU_SysCom_Transport
  VAR
    FB_SysCom_Transport : FB_Modbus_RTU_SysCom_Transport;
  END_VAR

            // ======================================================
// MODBUS RTU SYSCOM TRANSPORT EXECUTION
// ======================================================
// Byte-level transport boundary execution.
// ======================================================

FB_SysCom_Transport(
    VI_Enable := GVL_CONFIG.G_OpenTherm_Enabled,
    VI_System_Time_MS := GVL_STATUS.G_System_Time_MS
);
          
END_PROGRAM

PROGRAM PRG_Modbus_Master
  VAR
    L_i : INT;
    L_Elapsed_MS : UDINT;
  END_VAR

            // ======================================================
// MODBUS MASTER RUNTIME SCHEDULER
// ======================================================
// Library-independent Modbus master scheduler.
// ======================================================

IF NOT GVL_CONFIG.G_OpenTherm_Enabled THEN

    GVL_MODBUS_MASTER.G_Master_Online := FALSE;
    GVL_MODBUS_MASTER.G_Master_Error := FALSE;

    GVL_MODBUS_MASTER.G_Active := FALSE;
    GVL_MODBUS_MASTER.G_Active_Index := 0;
    GVL_MODBUS_MASTER.G_Active_Sequence := 0;
    GVL_MODBUS_MASTER.G_Active_Start_MS := 0;
    GVL_MODBUS_MASTER.G_Active_Retry_Count := 0;

    FOR L_i := 1 TO 16 DO
        GVL_MODBUS_MASTER.G_Response[L_i].Busy := FALSE;
        GVL_MODBUS_MASTER.G_Response[L_i].Done := FALSE;
        GVL_MODBUS_MASTER.G_Response[L_i].Error := FALSE;
        GVL_MODBUS_MASTER.G_Response[L_i].Error_Code := 0;
    END_FOR;

    RETURN;
END_IF;

GVL_MODBUS_MASTER.G_Master_Online :=
    GVL_MODBUS_RTU_BRIDGE.G_Driver_Online;

GVL_MODBUS_MASTER.G_Master_Error :=
    GVL_MODBUS_RTU_BRIDGE.G_Driver_Error;

// ======================================================
// START NEW TRANSACTION
// ======================================================
IF NOT GVL_MODBUS_MASTER.G_Active THEN

    FOR L_i := 1 TO 16 DO

        IF GVL_MODBUS_MASTER.G_Request[L_i].Enable THEN

            GVL_MODBUS_MASTER.G_Active := TRUE;
            GVL_MODBUS_MASTER.G_Active_Index := L_i;
            GVL_MODBUS_MASTER.G_Active_Sequence :=
                GVL_MODBUS_MASTER.G_Request[L_i].Sequence;

            GVL_MODBUS_MASTER.G_Active_Start_MS :=
                GVL_STATUS.G_System_Time_MS;

            GVL_MODBUS_MASTER.G_Active_Retry_Count := 0;

            GVL_MODBUS_MASTER.G_Response[L_i].Busy := TRUE;
            GVL_MODBUS_MASTER.G_Response[L_i].Done := FALSE;
            GVL_MODBUS_MASTER.G_Response[L_i].Error := FALSE;
            GVL_MODBUS_MASTER.G_Response[L_i].Error_Code := 0;

            EXIT;

        END_IF;

    END_FOR;

END_IF;

// ======================================================
// ACTIVE TRANSACTION SUPERVISION
// ======================================================
IF GVL_MODBUS_MASTER.G_Active THEN

    L_i := GVL_MODBUS_MASTER.G_Active_Index;

    L_Elapsed_MS :=
        GVL_STATUS.G_System_Time_MS -
        GVL_MODBUS_MASTER.G_Active_Start_MS;

    IF GVL_MODBUS_MASTER.G_Response[L_i].Done OR
       GVL_MODBUS_MASTER.G_Response[L_i].Error THEN

        GVL_MODBUS_MASTER.G_Response[L_i].Busy := FALSE;

        GVL_MODBUS_MASTER.G_Active := FALSE;
        GVL_MODBUS_MASTER.G_Last_Transaction_MS :=
            GVL_STATUS.G_System_Time_MS;

        GVL_MODBUS_MASTER.G_Total_Transactions :=
            GVL_MODBUS_MASTER.G_Total_Transactions + 1;

        IF GVL_MODBUS_MASTER.G_Response[L_i].Error THEN
            GVL_MODBUS_MASTER.G_Total_Errors :=
                GVL_MODBUS_MASTER.G_Total_Errors + 1;
        END_IF;

    ELSIF L_Elapsed_MS > GVL_MODBUS_MASTER.G_Request[L_i].Timeout_MS THEN

        GVL_MODBUS_MASTER.G_Active_Retry_Count :=
            GVL_MODBUS_MASTER.G_Active_Retry_Count + 1;

        IF GVL_MODBUS_MASTER.G_Active_Retry_Count >
           GVL_CONFIG.G_Modbus_RTU_Retry_Count THEN

            GVL_MODBUS_MASTER.G_Response[L_i].Busy := FALSE;
            GVL_MODBUS_MASTER.G_Response[L_i].Done := FALSE;
            GVL_MODBUS_MASTER.G_Response[L_i].Error := TRUE;
            GVL_MODBUS_MASTER.G_Response[L_i].Error_Code := 16#0003;

            GVL_MODBUS_MASTER.G_Response[L_i].Last_Sequence :=
                GVL_MODBUS_MASTER.G_Active_Sequence;

            GVL_MODBUS_MASTER.G_Response[L_i].Last_Update_MS :=
                GVL_STATUS.G_System_Time_MS;

            GVL_MODBUS_MASTER.G_Active := FALSE;

            GVL_MODBUS_MASTER.G_Total_Timeouts :=
                GVL_MODBUS_MASTER.G_Total_Timeouts + 1;

            GVL_MODBUS_MASTER.G_Total_Errors :=
                GVL_MODBUS_MASTER.G_Total_Errors + 1;

        ELSE

            GVL_MODBUS_MASTER.G_Active_Start_MS :=
                GVL_STATUS.G_System_Time_MS;

        END_IF;

    END_IF;

END_IF;
          
END_PROGRAM

PROGRAM PRG_Recovery_Ordering_Integrity_Governor

            IF GVL_DETERMINISTIC_RECOVERY_PATH_FABRIC.Deterministic_Recovery_Path_Granted
AND NOT GVL_RECOVERY_ORDERING_INTEGRITY_FABRIC.Unsafe_Recovery_Reordering_Detected
AND NOT GVL_RECOVERY_ORDERING_INTEGRITY_FABRIC.CrossDomain_Reactivation_Race
AND NOT GVL_RECOVERY_ORDERING_INTEGRITY_FABRIC.Recovery_Topology_Divergence
AND NOT GVL_RECOVERY_ORDERING_INTEGRITY_FABRIC.Residual_Unsafe_Reactivation_Detected THEN

    GVL_RECOVERY_ORDERING_INTEGRITY_FABRIC.Recovery_Ordering_Integrity_Valid := TRUE;
    GVL_RECOVERY_ORDERING_INTEGRITY_FABRIC.CrossDomain_Recovery_Ordering_Stable := TRUE;
    GVL_RECOVERY_ORDERING_INTEGRITY_FABRIC.Recovery_Authority_Sequencing_Canonical := TRUE;
    GVL_RECOVERY_ORDERING_INTEGRITY_FABRIC.Physical_Reactivation_Topology_Safe := TRUE;
END_IF;
          
END_PROGRAM

PROGRAM PRG_Forensic_Evidence_Governor
  VAR
    L_Now_MS : UDINT;
    L_Forensic_Valid : BOOL := TRUE;
    L_Error_Code : UDINT := 0;
    L_Error_Text : STRING(160) := '';
  END_VAR

            L_Now_MS := GVL_STATUS.G_System_Time_MS;
L_Forensic_Valid := TRUE;
L_Error_Code := 0;
L_Error_Text := '';

// Fail-safe defaults.
GVL_FORENSIC_EVIDENCE_FABRIC.Forensic_Evidence_Valid := FALSE;
GVL_FORENSIC_EVIDENCE_FABRIC.Forensic_Evidence_Granted := FALSE;
GVL_FORENSIC_EVIDENCE_FABRIC.Forensic_Evidence_Quarantine_Active := TRUE;

GVL_FORENSIC_EVIDENCE_FABRIC.Authority_Lineage_Reconstructable := FALSE;
GVL_FORENSIC_EVIDENCE_FABRIC.Decision_Causality_Traceable := FALSE;
GVL_FORENSIC_EVIDENCE_FABRIC.Distributed_Evidence_Coherent := FALSE;
GVL_FORENSIC_EVIDENCE_FABRIC.Immutable_Audit_Continuity_Valid := FALSE;
GVL_FORENSIC_EVIDENCE_FABRIC.Recovery_Lineage_Preserved := FALSE;

// Compliance federation required.
IF NOT GVL_COMPLIANCE_FEDERATION_FABRIC.Compliance_Federation_Granted THEN
    L_Forensic_Valid := FALSE;
    L_Error_Code := 43000;
    L_Error_Text := 'Compliance federation authority not granted';
END_IF;

// Forensic split-brain detectors.
IF GVL_FORENSIC_EVIDENCE_FABRIC.Authority_Lineage_Gap_Detected THEN
    L_Forensic_Valid := FALSE;
    L_Error_Code := 43001;
    L_Error_Text := 'Authority lineage gap detected';
END_IF;

IF GVL_FORENSIC_EVIDENCE_FABRIC.NonReconstructable_Decision_Detected THEN
    L_Forensic_Valid := FALSE;
    L_Error_Code := 43002;
    L_Error_Text := 'Non-reconstructable decision detected';
END_IF;

IF GVL_FORENSIC_EVIDENCE_FABRIC.History_Evidence_Divergence_Detected THEN
    L_Forensic_Valid := FALSE;
    L_Error_Code := 43003;
    L_Error_Text := 'History evidence divergence detected';
END_IF;

IF GVL_FORENSIC_EVIDENCE_FABRIC.Causal_Chain_Erosion_Detected THEN
    L_Forensic_Valid := FALSE;
    L_Error_Code := 43004;
    L_Error_Text := 'Causal chain erosion detected';
END_IF;

IF GVL_FORENSIC_EVIDENCE_FABRIC.Distributed_Forensic_Inconsistency_Detected THEN
    L_Forensic_Valid := FALSE;
    L_Error_Code := 43005;
    L_Error_Text := 'Distributed forensic inconsistency detected';
END_IF;

IF GVL_FORENSIC_EVIDENCE_FABRIC.Immutable_Audit_Discontinuity_Detected THEN
    L_Forensic_Valid := FALSE;
    L_Error_Code := 43006;
    L_Error_Text := 'Immutable audit discontinuity detected';
END_IF;

// Forensic reconstruction validation.
IF L_Forensic_Valid
AND NOT GVL_FORENSIC_EVIDENCE_FABRIC.Historical_Proof_Chain_Valid THEN
    L_Forensic_Valid := FALSE;
    L_Error_Code := 43010;
    L_Error_Text := 'Historical proof chain invalid';
END_IF;

IF L_Forensic_Valid
AND NOT GVL_FORENSIC_EVIDENCE_FABRIC.Governance_Event_Lineage_Coherent THEN
    L_Forensic_Valid := FALSE;
    L_Error_Code := 43011;
    L_Error_Text := 'Governance event lineage coherence invalid';
END_IF;

IF L_Forensic_Valid
AND NOT GVL_FORENSIC_EVIDENCE_FABRIC.Semantic_Transition_Traceable THEN
    L_Forensic_Valid := FALSE;
    L_Error_Code := 43012;
    L_Error_Text := 'Semantic transition traceability invalid';
END_IF;

IF L_Forensic_Valid
AND NOT GVL_FORENSIC_EVIDENCE_FABRIC.Physical_Transition_Traceable THEN
    L_Forensic_Valid := FALSE;
    L_Error_Code := 43013;
    L_Error_Text := 'Physical transition traceability invalid';
END_IF;

IF L_Forensic_Valid THEN
    GVL_FORENSIC_EVIDENCE_FABRIC.Forensic_Evidence_Valid := TRUE;
    GVL_FORENSIC_EVIDENCE_FABRIC.Forensic_Evidence_Granted := TRUE;
    GVL_FORENSIC_EVIDENCE_FABRIC.Forensic_Evidence_Quarantine_Active := FALSE;

    GVL_FORENSIC_EVIDENCE_FABRIC.Authority_Lineage_Reconstructable := TRUE;
    GVL_FORENSIC_EVIDENCE_FABRIC.Decision_Causality_Traceable := TRUE;
    GVL_FORENSIC_EVIDENCE_FABRIC.Distributed_Evidence_Coherent := TRUE;
    GVL_FORENSIC_EVIDENCE_FABRIC.Immutable_Audit_Continuity_Valid := TRUE;
    GVL_FORENSIC_EVIDENCE_FABRIC.Recovery_Lineage_Preserved := TRUE;

    GVL_FORENSIC_EVIDENCE_FABRIC.Forensic_Evidence_Epoch :=
        GVL_COMPLIANCE_FEDERATION_FABRIC.Compliance_Federation_Epoch;

    GVL_FORENSIC_EVIDENCE_FABRIC.Forensic_Evidence_Epoch_Coherent := TRUE;

    GVL_FORENSIC_EVIDENCE_FABRIC.Forensic_Evidence_Last_Update_MS :=
        L_Now_MS;

    GVL_FORENSIC_EVIDENCE_FABRIC.Forensic_Evidence_Lease_Expired := FALSE;

    GVL_FORENSIC_EVIDENCE_FABRIC.Forensic_Evidence_Last_Error_Code := 0;
    GVL_FORENSIC_EVIDENCE_FABRIC.Forensic_Evidence_Last_Error_Text := '';
ELSE
    GVL_FORENSIC_EVIDENCE_FABRIC.Forensic_Evidence_Valid := FALSE;
    GVL_FORENSIC_EVIDENCE_FABRIC.Forensic_Evidence_Granted := FALSE;
    GVL_FORENSIC_EVIDENCE_FABRIC.Forensic_Evidence_Quarantine_Active := TRUE;

    GVL_FORENSIC_EVIDENCE_FABRIC.Forensic_Evidence_Lease_Expired := TRUE;

    GVL_FORENSIC_EVIDENCE_FABRIC.Forensic_Evidence_Last_Error_Code :=
        L_Error_Code;

    GVL_FORENSIC_EVIDENCE_FABRIC.Forensic_Evidence_Last_Error_Text :=
        L_Error_Text;

    GVL_FORENSIC_EVIDENCE_FABRIC.Forensic_Evidence_Invalidation_Count :=
        GVL_FORENSIC_EVIDENCE_FABRIC.Forensic_Evidence_Invalidation_Count + 1;
END_IF;
          
END_PROGRAM

PROGRAM PRG_Runtime_Snapshot_Governor
  VAR
    L_Now_MS : UDINT;
    L_Snapshot_Valid : BOOL := TRUE;
    L_Error_Code : UDINT := 0;
    L_Error_Text : STRING(160) := '';
    L_Distributed_Publication_Healthy : BOOL;
  END_VAR

            L_Now_MS := GVL_STATUS.G_System_Time_MS;
L_Snapshot_Valid := TRUE;
L_Error_Code := 0;
L_Error_Text := '';

// ======================================================
// IMMUTABLE RUNTIME SNAPSHOT GOVERNOR
// ======================================================
// Governs immutable publication snapshot semantics.
// Prevents mutable runtime publication leakage.
//
// Runtime snapshot is upstream of output freshness.
// However distributed publication continuity must
// still remain semantically consistent.
// ======================================================

GVL_RUNTIME_SNAPSHOT.Snapshot_Mutation_Detected := FALSE;
GVL_RUNTIME_SNAPSHOT.Snapshot_Publication_Allowed := FALSE;
GVL_RUNTIME_SNAPSHOT.Snapshot_Frozen := FALSE;

// ------------------------------------------------------
// Runtime authority linkage.
// ------------------------------------------------------

IF NOT GVL_RUNTIME_EPOCH.Runtime_Runtime_Barrier_OK THEN
    L_Snapshot_Valid := FALSE;
    L_Error_Code := 12000;
    L_Error_Text := 'Runtime authority invalid';
END_IF;

// ------------------------------------------------------
// Distributed publication continuity linkage.
// ------------------------------------------------------

L_Distributed_Publication_Healthy :=
    GVL_DISTRIBUTED_SNAPSHOT.Distributed_Publication_Reconciled
    AND GVL_DISTRIBUTED_SNAPSHOT.Distributed_Publication_Freeze_Valid
    AND GVL_DISTRIBUTED_SNAPSHOT.Distributed_Snapshot_Consistent
    AND GVL_DISTRIBUTED_COMMIT.Distributed_Commit_Valid
    AND GVL_DISTRIBUTED_COMMIT.Publication_Prepare_Valid
    AND GVL_DISTRIBUTED_COMMIT.Publication_Commit_Confirmed
    AND NOT GVL_DISTRIBUTED_COMMIT.Peer_Commit_Mismatch
    AND NOT GVL_DISTRIBUTED_COMMIT.Commit_Lease_Expired;

IF L_Snapshot_Valid
AND NOT L_Distributed_Publication_Healthy
THEN
    L_Snapshot_Valid := FALSE;
    L_Error_Code := 12001;
    L_Error_Text := 'Distributed publication continuity invalid';
END_IF;

// ------------------------------------------------------
// Mutation detection foundation.
// ------------------------------------------------------

IF L_Snapshot_Valid
AND GVL_RUNTIME_EPOCH.Runtime_Impossible_State_Detected
THEN
    L_Snapshot_Valid := FALSE;
    L_Error_Code := 12003;
    L_Error_Text := 'Runtime mutation anomaly detected';

    GVL_RUNTIME_SNAPSHOT.Snapshot_Mutation_Detected := TRUE;
END_IF;

// ------------------------------------------------------
// Immutable snapshot freeze semantics.
// ------------------------------------------------------

IF L_Snapshot_Valid THEN
    GVL_RUNTIME_SNAPSHOT.Snapshot_Frozen := TRUE;
    GVL_RUNTIME_SNAPSHOT.Snapshot_Publication_Allowed := TRUE;

    GVL_RUNTIME_SNAPSHOT.Snapshot_Copy_Valid := TRUE;
    GVL_RUNTIME_SNAPSHOT.Snapshot_Isolation_Valid := TRUE;

    GVL_RUNTIME_SNAPSHOT.Snapshot_Runtime_Authority_Valid := TRUE;

    GVL_RUNTIME_SNAPSHOT.Snapshot_Freeze_Start_MS := L_Now_MS;
    GVL_RUNTIME_SNAPSHOT.Snapshot_Last_Publication_MS := L_Now_MS;

    GVL_RUNTIME_SNAPSHOT.Snapshot_Epoch := GVL_RUNTIME_SNAPSHOT.Snapshot_Epoch + 1;
    GVL_RUNTIME_SNAPSHOT.Snapshot_Publication_Epoch := GVL_RUNTIME_SNAPSHOT.Snapshot_Publication_Epoch + 1;

    GVL_RUNTIME_SNAPSHOT.Snapshot_Last_Error_Code := 0;
    GVL_RUNTIME_SNAPSHOT.Snapshot_Last_Error_Text := '';
ELSE
    GVL_RUNTIME_SNAPSHOT.Snapshot_Frozen := FALSE;
    GVL_RUNTIME_SNAPSHOT.Snapshot_Publication_Allowed := FALSE;

    GVL_RUNTIME_SNAPSHOT.Snapshot_Copy_Valid := FALSE;
    GVL_RUNTIME_SNAPSHOT.Snapshot_Isolation_Valid := FALSE;

    GVL_RUNTIME_SNAPSHOT.Snapshot_Runtime_Authority_Valid := FALSE;

    GVL_RUNTIME_SNAPSHOT.Snapshot_Last_Error_Code := L_Error_Code;
    GVL_RUNTIME_SNAPSHOT.Snapshot_Last_Error_Text := L_Error_Text;
END_IF;
          
END_PROGRAM

PROGRAM PRG_Config_Validation
  VAR
    fbConfigSimulation : FB_Config_Simulation;
    L_i : INT;
    L_Zone : INT;
    L_Sensor : INT;
    L_Manifold : INT;
    L_Map_Index : INT;
    L_Config_Error : BOOL;
  END_VAR

            // ======================================================
// CENTRAL CONFIGURATION VALIDATION
// ======================================================
// Diagnostic-only layer.
//
// This PRG may set validation/configuration status flags and text,
// but must not directly mutate aggregated diagnostics fields.
// Aggregated diagnostics ownership is centralized in:
//
//   FB_System_Health_Orchestrator
//
// This PRG also must not write command/shadow/output structures.
// ======================================================

L_Config_Error := FALSE;

// ======================================================
// ACTIVE SIZE CONFIGURATION
// ======================================================
IF (GVL_SYSTEM_SIZE_CONFIG.G_Active_Heating_Circuits < 1) OR
   (GVL_SYSTEM_SIZE_CONFIG.G_Active_Heating_Circuits > GVL_CONSTANTS.C_MAX_HEATING_CIRCUITS) THEN
    L_Config_Error := TRUE;
END_IF;

IF (GVL_SYSTEM_SIZE_CONFIG.G_Active_Water_Zones < 1) OR
   (GVL_SYSTEM_SIZE_CONFIG.G_Active_Water_Zones > GVL_CONSTANTS.C_MAX_WATER_ZONES) THEN
    L_Config_Error := TRUE;
END_IF;

IF (GVL_SYSTEM_SIZE_CONFIG.G_Active_Light_Zones < 1) OR
   (GVL_SYSTEM_SIZE_CONFIG.G_Active_Light_Zones > GVL_CONSTANTS.C_MAX_LIGHT_ZONES) THEN
    L_Config_Error := TRUE;
END_IF;

IF (GVL_SYSTEM_SIZE_CONFIG.G_Active_Blinds < 0) OR
   (GVL_SYSTEM_SIZE_CONFIG.G_Active_Blinds > GVL_CONSTANTS.C_MAX_BLINDS) THEN
    L_Config_Error := TRUE;
END_IF;

IF (GVL_SYSTEM_SIZE_CONFIG.G_Active_Sockets < 0) OR
   (GVL_SYSTEM_SIZE_CONFIG.G_Active_Sockets > GVL_CONSTANTS.C_MAX_SOCKETS) THEN
    L_Config_Error := TRUE;
END_IF;

// ======================================================
// HEATING CIRCUIT CONFIGURATION
// ======================================================
FOR L_i := 1 TO GVL_CONSTANTS.C_MAX_HEATING_CIRCUITS DO
    L_Zone := BYTE_TO_INT(GVL_CONFIG.G_HMI_FloorHeating_Configs[L_i].zone);
    L_Sensor := BYTE_TO_INT(GVL_CONFIG.G_HMI_FloorHeating_Configs[L_i].sensor_id);
    L_Manifold := BYTE_TO_INT(GVL_CONFIG.G_HMI_FloorHeating_Configs[L_i].manifold_id);

    IF (L_Zone < 1) OR (L_Zone > GVL_CONSTANTS.C_MAX_ZONES) THEN
        L_Config_Error := TRUE;
    END_IF;

    IF (L_Sensor < 1) OR (L_Sensor > GVL_CONSTANTS.C_MAX_ZONES) THEN
        L_Config_Error := TRUE;
    END_IF;

    IF (L_Manifold < 1) OR (L_Manifold > GVL_CONSTANTS.C_MAX_MANIFOLDS) THEN
        L_Config_Error := TRUE;
    END_IF;

    IF GVL_CONFIG.G_HMI_FloorHeating_Configs[L_i].min_temp > GVL_CONFIG.G_HMI_FloorHeating_Configs[L_i].max_temp THEN
        L_Config_Error := TRUE;
    END_IF;
END_FOR;

IF (GVL_CONFIG.G_Max_Active_Manifolds < 1) OR
   (GVL_CONFIG.G_Max_Active_Manifolds > GVL_CONSTANTS.C_MAX_MANIFOLDS) THEN
    L_Config_Error := TRUE;
END_IF;

IF GVL_CONFIG.G_Max_Thermal_Budget <= 0.0 THEN
    L_Config_Error := TRUE;
END_IF;

IF GVL_CONFIG.G_Policy_Min_Hold_MS < 10000 THEN
    L_Config_Error := TRUE;
END_IF;

// ======================================================
// ACCESS / TIMING CONFIGURATION
// ======================================================
IF (GVL_CONFIG.G_Access_Pulse_MS < 100) OR (GVL_CONFIG.G_Access_Pulse_MS > 5000) THEN
    L_Config_Error := TRUE;
END_IF;

// ======================================================
// MAP CONFIGURATION
// ======================================================
FOR L_i := 1 TO GVL_CONSTANTS.C_MAX_DOOR_SENSORS DO
    L_Map_Index := GVL_CONFIG.G_Door_Map[L_i];
    IF (L_Map_Index < 1) OR (L_Map_Index > GVL_CONSTANTS.C_MAX_SECURITY_SENSORS) THEN
        L_Config_Error := TRUE;
    END_IF;
END_FOR;

FOR L_i := 1 TO GVL_CONSTANTS.C_MAX_ZONES DO
    L_Map_Index := GVL_CONFIG.G_Window_Map[L_i];
    IF L_Map_Index <> 0 THEN
        IF (L_Map_Index < 1) OR (L_Map_Index > (GVL_CONSTANTS.C_MAX_SECURITY_SENSORS * 2)) THEN
            L_Config_Error := TRUE;
        END_IF;
    END_IF;
END_FOR;

FOR L_i := 1 TO GVL_CONSTANTS.C_MAX_HEATING_CIRCUITS DO
    IF (GVL_CONFIG.G_FloorTemp_Map[L_i] < 1) OR (GVL_CONFIG.G_FloorTemp_Map[L_i] > GVL_CONSTANTS.C_MAX_ZONES) THEN
        L_Config_Error := TRUE;
    END_IF;
END_FOR;

FOR L_i := 1 TO GVL_CONSTANTS.C_MAX_ZONES DO
    IF (GVL_CONFIG.G_RoomTemp_Map[L_i] < 1) OR (GVL_CONFIG.G_RoomTemp_Map[L_i] > GVL_CONSTANTS.C_MAX_ZONES) THEN
        L_Config_Error := TRUE;
    END_IF;
END_FOR;

// ======================================================
// HARDWARE SERVICE / RETRY CONFIGURATION
// ======================================================
IF GVL_CONFIG.G_Freeze_Hardware_Retry_Count < 0 THEN
    L_Config_Error := TRUE;
END_IF;

IF GVL_CONFIG.G_Freeze_Hardware_Retry_Delay_MS < 1000 THEN
    L_Config_Error := TRUE;
END_IF;

IF GVL_CONFIG.G_Pump_Exercise_Enabled THEN
    IF GVL_CONFIG.G_Pump_Exercise_Interval_MS < GVL_CONSTANTS.C_MS_IN_MINUTE THEN
        L_Config_Error := TRUE;
    END_IF;
    IF GVL_CONFIG.G_Pump_Exercise_Duration_MS < 1000 THEN
        L_Config_Error := TRUE;
    END_IF;
END_IF;

IF GVL_CONFIG.G_Water_Valve_Exercise_Enabled THEN
    IF GVL_CONFIG.G_Water_Valve_Exercise_Interval_MS < GVL_CONSTANTS.C_MS_IN_MINUTE THEN
        L_Config_Error := TRUE;
    END_IF;
    IF GVL_CONFIG.G_Water_Valve_Exercise_Duration_MS < 1000 THEN
        L_Config_Error := TRUE;
    END_IF;
END_IF;

IF GVL_CONFIG.G_Water_Valve_Close_Retry_Count < 0 THEN
    L_Config_Error := TRUE;
END_IF;

IF GVL_CONFIG.G_Water_Valve_Close_Retry_Delay_MS < 1000 THEN
    L_Config_Error := TRUE;
END_IF;

// ======================================================
// OPENTHERM / MODBUS RTU CONFIGURATION
// ======================================================
IF GVL_CONFIG.G_OpenTherm_Enabled THEN

    IF GVL_CONFIG.G_OpenTherm_Heartbeat_Timeout_MS < 1000 THEN
        L_Config_Error := TRUE;
    END_IF;

    IF GVL_CONFIG.G_OpenTherm_Command_Ack_Timeout_MS < 500 THEN
        L_Config_Error := TRUE;
    END_IF;

    IF GVL_CONFIG.G_Modbus_RTU_Baudrate < 1200 THEN
        L_Config_Error := TRUE;
    END_IF;

    IF (GVL_CONFIG.G_Modbus_RTU_Parity > 2) THEN
        L_Config_Error := TRUE;
    END_IF;

    IF (GVL_CONFIG.G_Modbus_RTU_Stop_Bits < 1) OR
       (GVL_CONFIG.G_Modbus_RTU_Stop_Bits > 2) THEN
        L_Config_Error := TRUE;
    END_IF;

    IF (GVL_CONFIG.G_Modbus_RTU_Data_Bits < 7) OR
       (GVL_CONFIG.G_Modbus_RTU_Data_Bits > 8) THEN
        L_Config_Error := TRUE;
    END_IF;

    IF GVL_CONFIG.G_Modbus_RTU_Slave_ID = 0 THEN
        L_Config_Error := TRUE;
    END_IF;

    IF GVL_CONFIG.G_Modbus_RTU_Poll_Interval_MS < 50 THEN
        L_Config_Error := TRUE;
    END_IF;

    IF GVL_CONFIG.G_Modbus_RTU_Request_Timeout_MS < 50 THEN
        L_Config_Error := TRUE;
    END_IF;

    IF GVL_CONFIG.G_Modbus_RTU_Retry_Count < 0 THEN
        L_Config_Error := TRUE;
    END_IF;

    FOR L_i := 1 TO GVL_CONSTANTS.C_MAX_BOILERS DO
        IF GVL_CONFIG.G_OpenTherm_Register_Map[L_i].Cmd_Enable_Offset = GVL_CONFIG.G_OpenTherm_Register_Map[L_i].Status_Word_Offset THEN
            L_Config_Error := TRUE;
        END_IF;

        IF GVL_CONFIG.G_OpenTherm_Register_Map[L_i].Cmd_Setpoint_x10_Offset = GVL_CONFIG.G_OpenTherm_Register_Map[L_i].Status_Word_Offset THEN
            L_Config_Error := TRUE;
        END_IF;
    END_FOR;
END_IF;

// ======================================================
// SENSOR COUNT SANITY
// ======================================================
IF GVL_CONSTANTS.C_MAX_METHANE_SENSORS < 2 THEN
    L_Config_Error := TRUE;
END_IF;

IF GVL_CONSTANTS.C_MAX_SMOKE_SENSORS < 6 THEN
    L_Config_Error := TRUE;
END_IF;

IF GVL_CONSTANTS.C_MAX_CO_SENSORS < 8 THEN
    L_Config_Error := TRUE;
END_IF;

IF GVL_CONSTANTS.C_MAX_FLOOD_SENSORS < 9 THEN
    L_Config_Error := TRUE;
END_IF;

// ======================================================
// CONFIG SIMULATION / COMMISSIONING VALIDATION
// ======================================================
fbConfigSimulation(
    VI_Enable := TRUE,
    VI_Request := GVL_CONFIG_SIMULATION.G_Simulation_Request,
    VI_Confirm := GVL_CONFIG_SIMULATION.G_Simulation_Confirm
);

IF fbConfigSimulation.VO_Executed AND NOT fbConfigSimulation.VO_Result_OK THEN
    L_Config_Error := TRUE;
END_IF;

